// TIA Portal V20 program export: 0 tag tables, 2 data types, 3 data blocks, 7 code blocks (in call order from the OBs), 3 instance data blocks

TYPE "UDT_PusherIO"
// stored: IsFailsafeCompliant false
   STRUCT
      "Step" : Int;
      Fitted : Bool;
      Enable : Bool;
      Mode : Int;
      HopperHighLevel : Bool;
      ManualCycleCmd : Bool;
      JogExtendCmd : Bool;
      JogRetractCmd : Bool;
      HomeLimit : Bool;
      FullTravelLimit : Bool;
      HighPressure : Bool;
      PowerPackRunningFB : Bool;
      FaultReset : Bool;
      EndTravelTimeout : Real;
      ParkedTimeout : Real;
      EndTravelHoldTime : Real;
      PumpRunOnTime : Real;
      JogWarningTime : Real;
      PressureTripConfirmTime : Real;
      PressureClearResumeDelay : Real;
      PressureTripCountThreshold : Int;
      Cycling : Bool;
      Blocked : Bool;
      EndTravelTimeoutFault : Bool;
      ParkedTimeoutFault : Bool;
      BothSwitchesFault : Bool;
      RunPowerPack : Bool;
      Extend : Bool;
      Retract : Bool;
      JogPreStartSounder : Bool;
   END_STRUCT;
END_TYPE

TYPE "UDT_ShredderSequencerIO"
// stored: IsFailsafeCompliant false
   STRUCT
      CycleStart : Bool;
      CycleStop : Bool;
      DownstreamRunning : Bool;
      DischargeConvRunning : Bool;
      HopperLevelHigh : Bool;
      ShredderRunFwdFB : Bool;
      ShredderMotorCurrent : Real;
      MotorFaultActive : Bool;
      FaultReset : Bool;
      OperatorPusherMode : Int;
      PusherJogPreStartSounder : Bool;
      "Step" : Int;
      DischargeConveyorTimeoutFault : Bool;
      ShredderBlockedFault : Bool;
      RunDischargeConv : Bool;
      RunInfeedConv : Bool;
      EnableUpstream : Bool;
      PreStartSounder : Bool;
      InCycle : Bool;
      MotorReverseCmd : Bool;
      MotorAutoStartCmd : Bool;
      MotorPreStartDoneCmd : Bool;
      PusherModeCmd : Int;
   END_STRUCT;
END_TYPE

DATA_BLOCK "DB_Alarms"   // DB5
{ S7_Optimized_Access := 'TRUE' }
VERSION : 0.1
// Category alarms packed per Word (C-501). Bits written by FC_AlarmsMain via documented slice-access exception to C-301.
// stored: AutoNumber true, DBAccessibleFromOPCUA true, IsOnlyStoredInLoadMemory false, IsRetainMemResEnabled false, IsWriteProtectedInAS false, MemoryReserve 100
   VAR
      ShredderAlarm0 : Word;
   END_VAR
BEGIN
END_DATA_BLOCK

DATA_BLOCK "DB_Output"   // DB2
{ S7_Optimized_Access := 'TRUE' }
VERSION : 0.1
// stored: AutoNumber true, DBAccessibleFromOPCUA true, IsOnlyStoredInLoadMemory false, IsRetainMemResEnabled false, IsWriteProtectedInAS false, MemoryReserve 100
   VAR
      Test : Array[0..18] of Bool;
      SpareDQ : Array[1..7] of Bool;
      Run_Shredder_Fwd : Bool;
      Run_Shredder_Rev : Bool;
      Run_PowerPack : Bool;
      Run_Infeed_Conv : Bool;
      Run_Discharge_Conv : Bool;
      Pusher_Extend : Bool;
      Pusher_Retract : Bool;
      In_Cycle : Bool;
      Enable_Upstream : Bool;
      PreStart_Sounder : Bool;
      Motor_Fault_Reset : Bool;
   END_VAR
BEGIN
END_DATA_BLOCK

DATA_BLOCK "DB_Settings"   // DB3
{ S7_Optimized_Access := 'TRUE' }
VERSION : 0.1
// Plant/system-level tunables (C-307) - HMI/operator writes, PLC read-only (C-308). Start values are commissioning defaults (C-309). Members with no start value shown are genuinely unconfigured pending real numbers from the project owner - see the presented build notes, not a guess.
// stored: AutoNumber true, DBAccessibleFromOPCUA true, IsOnlyStoredInLoadMemory false, IsRetainMemResEnabled false, IsWriteProtectedInAS false, MemoryReserve 100
   VAR RETAIN
      PreStartSounderTime : Real := 10.0;
      ShredderReverseRunTime : Real := 6.0;
      InfeedRestartDelay : Real := 5.0;
      InfeedToUpstreamEnableDelay : Real := 3.0;
      OvercurrentSetpointMedium : Real;
      OvercurrentSetpointHigh : Real;
      OvercurrentMediumDelay : Real;
      OvercurrentHighDelay : Real;
      OvercurrentSpinUpAllowance : Real := 3.0;
      ReversalRetryPauseTime : Real := 4.0;
      ReversalWindowTime : Real := 180.0;
      ReversalCountThreshold : Int := 5;
      PressureTripConfirmTime : Real := 0.5;
      PressureClearResumeDelay : Real;
      PressureTripCountThreshold : Int := 5;
      PusherEndTravelTimeout : Real;
      PusherParkedTimeout : Real;
      PusherEndTravelHoldTime : Real := 2.0;
      PusherPumpRunOnTime : Real;
      PusherJogWarningTime : Real := 1.0;
      PusherFitted : Bool := TRUE;
      DischargeConveyorTimeout : Real;
   END_VAR
BEGIN
END_DATA_BLOCK

ORGANIZATION_BLOCK "Main"   // OB1, LAD, ProgramCycle
TITLE = "Main Program Sweep (Cycle)"
{ S7_Optimized_Access := 'TRUE' }
VERSION : 0.1
// stored: AutoNumber true, IsIECCheckEnabled false, SetENOAutomatically false
   VAR_INPUT
      Initial_Call : Bool;   // Initial call of this OB
      Remanence : Bool;   // =True, if remanent data are available
   END_VAR
BEGIN

REGION Network 1: Input Mapping
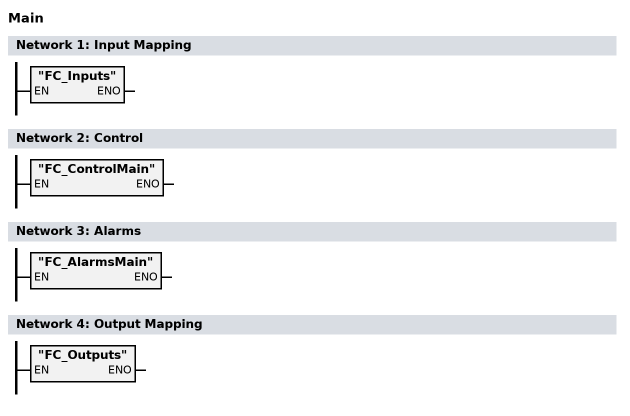
   RUNG wire#powerrail
      "FC_Inputs"()
   END_RUNG
   // the same network as SCL:
   "FC_Inputs"();
END_REGION

REGION Network 2: Control
   RUNG wire#powerrail
      "FC_ControlMain"()
   END_RUNG
   // the same network as SCL:
   "FC_ControlMain"();
END_REGION

REGION Network 3: Alarms
   RUNG wire#powerrail
      "FC_AlarmsMain"()
   END_RUNG
   // the same network as SCL:
   "FC_AlarmsMain"();
END_REGION

REGION Network 4: Output Mapping
   RUNG wire#powerrail
      "FC_Outputs"()
   END_RUNG
   // the same network as SCL:
   "FC_Outputs"();
END_REGION
END_ORGANIZATION_BLOCK

FUNCTION "FC_Inputs" : Void   // FC1, LAD
TITLE = Input Map
{ S7_Optimized_Access := 'TRUE' }
VERSION : 0.1
// stored: AutoNumber true, IsIECCheckEnabled false, SetENOAutomatically false, UDAEnableTagReadback false
BEGIN

REGION Network 1: PLC1 Built-in DI (CPU 1214C)
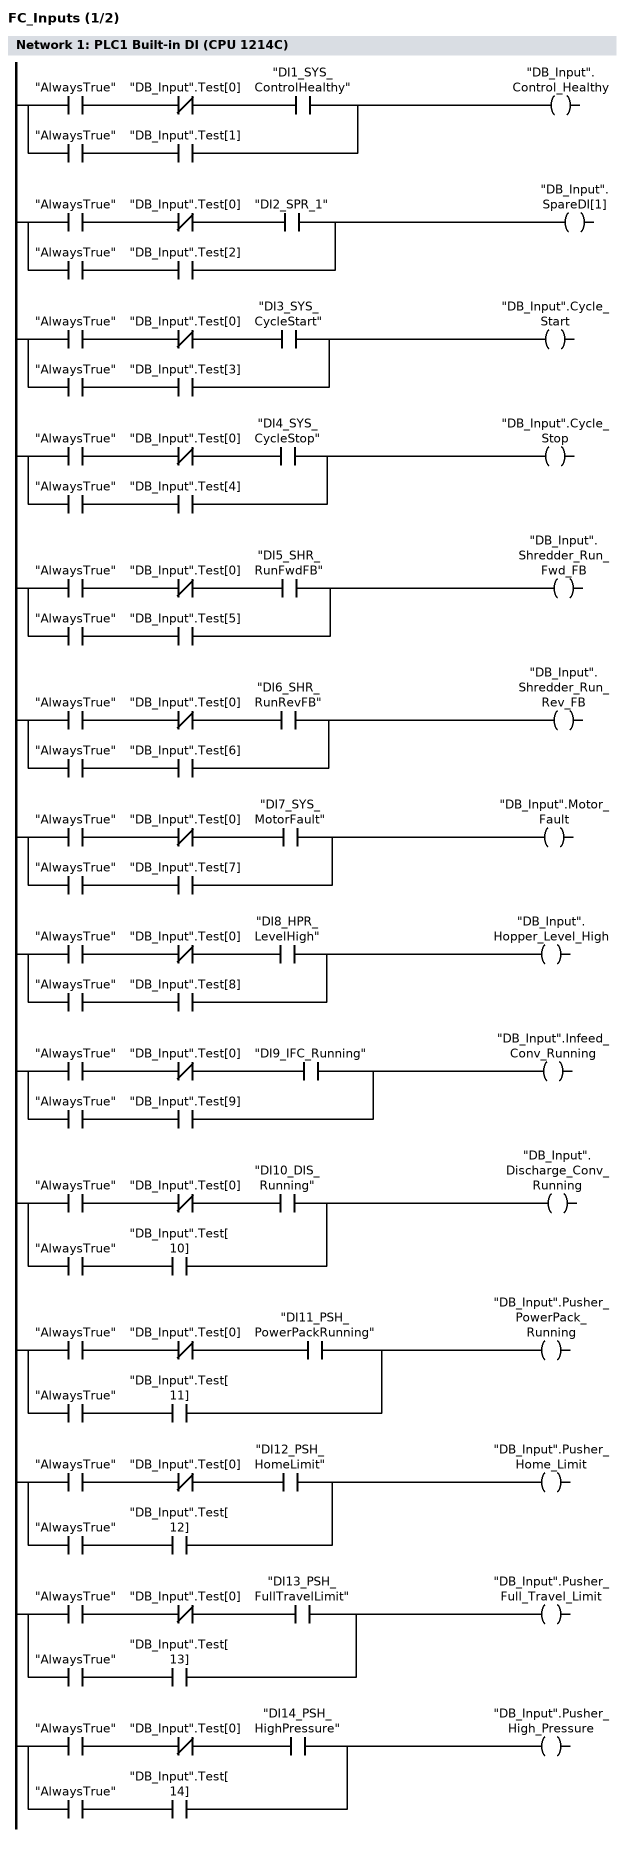
   RUNG wire#powerrail
      Contact( "AlwaysTrue" )
      I_Contact( "DB_Input".Test[0] )
      Contact( "DI1_SYS_ControlHealthy" )
      wire#w1
      Coil( "DB_Input".Control_Healthy )
   END_RUNG
   RUNG wire#powerrail
      Contact( "AlwaysTrue" )
      Contact( "DB_Input".Test[1] )
   END_RUNG wire#w1
   RUNG wire#powerrail
      Contact( "AlwaysTrue" )
      I_Contact( "DB_Input".Test[0] )
      Contact( "DI2_SPR_1" )
      wire#w2
      Coil( "DB_Input".SpareDI[1] )
   END_RUNG
   RUNG wire#powerrail
      Contact( "AlwaysTrue" )
      Contact( "DB_Input".Test[2] )
   END_RUNG wire#w2
   RUNG wire#powerrail
      Contact( "AlwaysTrue" )
      I_Contact( "DB_Input".Test[0] )
      Contact( "DI3_SYS_CycleStart" )
      wire#w3
      Coil( "DB_Input".Cycle_Start )
   END_RUNG
   RUNG wire#powerrail
      Contact( "AlwaysTrue" )
      Contact( "DB_Input".Test[3] )
   END_RUNG wire#w3
   RUNG wire#powerrail
      Contact( "AlwaysTrue" )
      I_Contact( "DB_Input".Test[0] )
      Contact( "DI4_SYS_CycleStop" )
      wire#w4
      Coil( "DB_Input".Cycle_Stop )
   END_RUNG
   RUNG wire#powerrail
      Contact( "AlwaysTrue" )
      Contact( "DB_Input".Test[4] )
   END_RUNG wire#w4
   RUNG wire#powerrail
      Contact( "AlwaysTrue" )
      I_Contact( "DB_Input".Test[0] )
      Contact( "DI5_SHR_RunFwdFB" )
      wire#w5
      Coil( "DB_Input".Shredder_Run_Fwd_FB )
   END_RUNG
   RUNG wire#powerrail
      Contact( "AlwaysTrue" )
      Contact( "DB_Input".Test[5] )
   END_RUNG wire#w5
   RUNG wire#powerrail
      Contact( "AlwaysTrue" )
      I_Contact( "DB_Input".Test[0] )
      Contact( "DI6_SHR_RunRevFB" )
      wire#w6
      Coil( "DB_Input".Shredder_Run_Rev_FB )
   END_RUNG
   RUNG wire#powerrail
      Contact( "AlwaysTrue" )
      Contact( "DB_Input".Test[6] )
   END_RUNG wire#w6
   RUNG wire#powerrail
      Contact( "AlwaysTrue" )
      I_Contact( "DB_Input".Test[0] )
      Contact( "DI7_SYS_MotorFault" )
      wire#w7
      Coil( "DB_Input".Motor_Fault )
   END_RUNG
   RUNG wire#powerrail
      Contact( "AlwaysTrue" )
      Contact( "DB_Input".Test[7] )
   END_RUNG wire#w7
   RUNG wire#powerrail
      Contact( "AlwaysTrue" )
      I_Contact( "DB_Input".Test[0] )
      Contact( "DI8_HPR_LevelHigh" )
      wire#w8
      Coil( "DB_Input".Hopper_Level_High )
   END_RUNG
   RUNG wire#powerrail
      Contact( "AlwaysTrue" )
      Contact( "DB_Input".Test[8] )
   END_RUNG wire#w8
   RUNG wire#powerrail
      Contact( "AlwaysTrue" )
      I_Contact( "DB_Input".Test[0] )
      Contact( "DI9_IFC_Running" )
      wire#w9
      Coil( "DB_Input".Infeed_Conv_Running )
   END_RUNG
   RUNG wire#powerrail
      Contact( "AlwaysTrue" )
      Contact( "DB_Input".Test[9] )
   END_RUNG wire#w9
   RUNG wire#powerrail
      Contact( "AlwaysTrue" )
      I_Contact( "DB_Input".Test[0] )
      Contact( "DI10_DIS_Running" )
      wire#w10
      Coil( "DB_Input".Discharge_Conv_Running )
   END_RUNG
   RUNG wire#powerrail
      Contact( "AlwaysTrue" )
      Contact( "DB_Input".Test[10] )
   END_RUNG wire#w10
   RUNG wire#powerrail
      Contact( "AlwaysTrue" )
      I_Contact( "DB_Input".Test[0] )
      Contact( "DI11_PSH_PowerPackRunning" )
      wire#w11
      Coil( "DB_Input".Pusher_PowerPack_Running )
   END_RUNG
   RUNG wire#powerrail
      Contact( "AlwaysTrue" )
      Contact( "DB_Input".Test[11] )
   END_RUNG wire#w11
   RUNG wire#powerrail
      Contact( "AlwaysTrue" )
      I_Contact( "DB_Input".Test[0] )
      Contact( "DI12_PSH_HomeLimit" )
      wire#w12
      Coil( "DB_Input".Pusher_Home_Limit )
   END_RUNG
   RUNG wire#powerrail
      Contact( "AlwaysTrue" )
      Contact( "DB_Input".Test[12] )
   END_RUNG wire#w12
   RUNG wire#powerrail
      Contact( "AlwaysTrue" )
      I_Contact( "DB_Input".Test[0] )
      Contact( "DI13_PSH_FullTravelLimit" )
      wire#w13
      Coil( "DB_Input".Pusher_Full_Travel_Limit )
   END_RUNG
   RUNG wire#powerrail
      Contact( "AlwaysTrue" )
      Contact( "DB_Input".Test[13] )
   END_RUNG wire#w13
   RUNG wire#powerrail
      Contact( "AlwaysTrue" )
      I_Contact( "DB_Input".Test[0] )
      Contact( "DI14_PSH_HighPressure" )
      wire#w14
      Coil( "DB_Input".Pusher_High_Pressure )
   END_RUNG
   RUNG wire#powerrail
      Contact( "AlwaysTrue" )
      Contact( "DB_Input".Test[14] )
   END_RUNG wire#w14
   // the same network as SCL:
   "DB_Input".Control_Healthy := ("AlwaysTrue" AND NOT "DB_Input".Test[0] AND "DI1_SYS_ControlHealthy") OR ("AlwaysTrue" AND "DB_Input".Test[1]);
   "DB_Input".SpareDI[1] := ("AlwaysTrue" AND NOT "DB_Input".Test[0] AND "DI2_SPR_1") OR ("AlwaysTrue" AND "DB_Input".Test[2]);
   "DB_Input".Cycle_Start := ("AlwaysTrue" AND NOT "DB_Input".Test[0] AND "DI3_SYS_CycleStart") OR ("AlwaysTrue" AND "DB_Input".Test[3]);
   "DB_Input".Cycle_Stop := ("AlwaysTrue" AND NOT "DB_Input".Test[0] AND "DI4_SYS_CycleStop") OR ("AlwaysTrue" AND "DB_Input".Test[4]);
   "DB_Input".Shredder_Run_Fwd_FB := ("AlwaysTrue" AND NOT "DB_Input".Test[0] AND "DI5_SHR_RunFwdFB") OR ("AlwaysTrue" AND "DB_Input".Test[5]);
   "DB_Input".Shredder_Run_Rev_FB := ("AlwaysTrue" AND NOT "DB_Input".Test[0] AND "DI6_SHR_RunRevFB") OR ("AlwaysTrue" AND "DB_Input".Test[6]);
   "DB_Input".Motor_Fault := ("AlwaysTrue" AND NOT "DB_Input".Test[0] AND "DI7_SYS_MotorFault") OR ("AlwaysTrue" AND "DB_Input".Test[7]);
   "DB_Input".Hopper_Level_High := ("AlwaysTrue" AND NOT "DB_Input".Test[0] AND "DI8_HPR_LevelHigh") OR ("AlwaysTrue" AND "DB_Input".Test[8]);
   "DB_Input".Infeed_Conv_Running := ("AlwaysTrue" AND NOT "DB_Input".Test[0] AND "DI9_IFC_Running") OR ("AlwaysTrue" AND "DB_Input".Test[9]);
   "DB_Input".Discharge_Conv_Running := ("AlwaysTrue" AND NOT "DB_Input".Test[0] AND "DI10_DIS_Running") OR ("AlwaysTrue" AND "DB_Input".Test[10]);
   "DB_Input".Pusher_PowerPack_Running := ("AlwaysTrue" AND NOT "DB_Input".Test[0] AND "DI11_PSH_PowerPackRunning") OR ("AlwaysTrue" AND "DB_Input".Test[11]);
   "DB_Input".Pusher_Home_Limit := ("AlwaysTrue" AND NOT "DB_Input".Test[0] AND "DI12_PSH_HomeLimit") OR ("AlwaysTrue" AND "DB_Input".Test[12]);
   "DB_Input".Pusher_Full_Travel_Limit := ("AlwaysTrue" AND NOT "DB_Input".Test[0] AND "DI13_PSH_FullTravelLimit") OR ("AlwaysTrue" AND "DB_Input".Test[13]);
   "DB_Input".Pusher_High_Pressure := ("AlwaysTrue" AND NOT "DB_Input".Test[0] AND "DI14_PSH_HighPressure") OR ("AlwaysTrue" AND "DB_Input".Test[14]);
END_REGION

REGION Network 2: PLC1.1 SM1223 DI
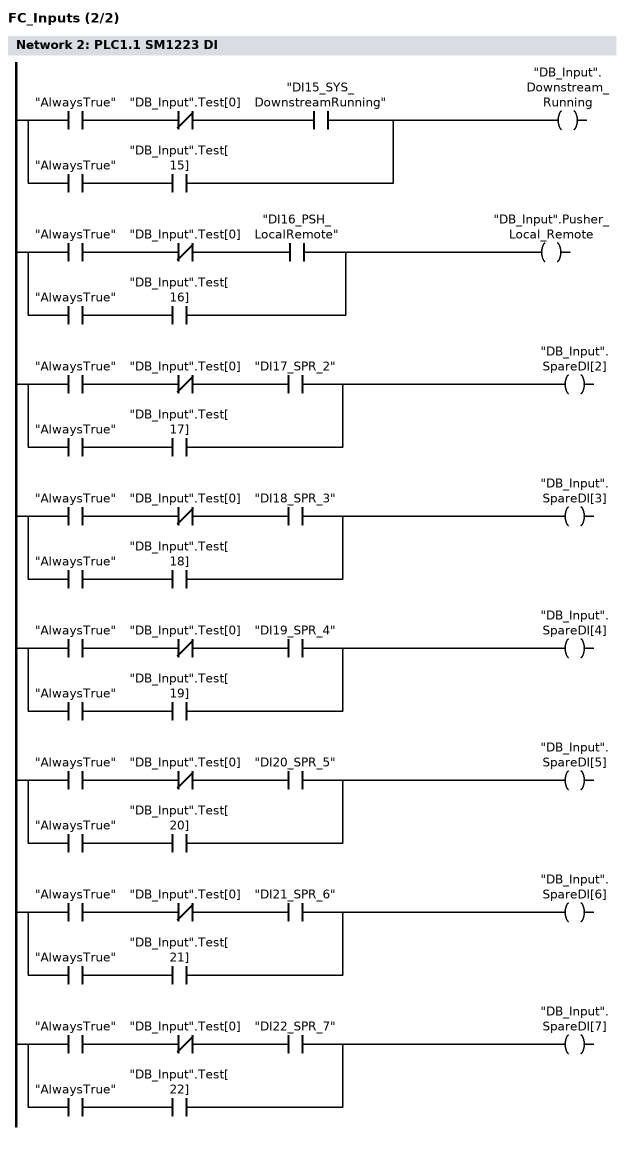
   RUNG wire#powerrail
      Contact( "AlwaysTrue" )
      I_Contact( "DB_Input".Test[0] )
      Contact( "DI15_SYS_DownstreamRunning" )
      wire#w1
      Coil( "DB_Input".Downstream_Running )
   END_RUNG
   RUNG wire#powerrail
      Contact( "AlwaysTrue" )
      Contact( "DB_Input".Test[15] )
   END_RUNG wire#w1
   RUNG wire#powerrail
      Contact( "AlwaysTrue" )
      I_Contact( "DB_Input".Test[0] )
      Contact( "DI16_PSH_LocalRemote" )
      wire#w2
      Coil( "DB_Input".Pusher_Local_Remote )
   END_RUNG
   RUNG wire#powerrail
      Contact( "AlwaysTrue" )
      Contact( "DB_Input".Test[16] )
   END_RUNG wire#w2
   RUNG wire#powerrail
      Contact( "AlwaysTrue" )
      I_Contact( "DB_Input".Test[0] )
      Contact( "DI17_SPR_2" )
      wire#w3
      Coil( "DB_Input".SpareDI[2] )
   END_RUNG
   RUNG wire#powerrail
      Contact( "AlwaysTrue" )
      Contact( "DB_Input".Test[17] )
   END_RUNG wire#w3
   RUNG wire#powerrail
      Contact( "AlwaysTrue" )
      I_Contact( "DB_Input".Test[0] )
      Contact( "DI18_SPR_3" )
      wire#w4
      Coil( "DB_Input".SpareDI[3] )
   END_RUNG
   RUNG wire#powerrail
      Contact( "AlwaysTrue" )
      Contact( "DB_Input".Test[18] )
   END_RUNG wire#w4
   RUNG wire#powerrail
      Contact( "AlwaysTrue" )
      I_Contact( "DB_Input".Test[0] )
      Contact( "DI19_SPR_4" )
      wire#w5
      Coil( "DB_Input".SpareDI[4] )
   END_RUNG
   RUNG wire#powerrail
      Contact( "AlwaysTrue" )
      Contact( "DB_Input".Test[19] )
   END_RUNG wire#w5
   RUNG wire#powerrail
      Contact( "AlwaysTrue" )
      I_Contact( "DB_Input".Test[0] )
      Contact( "DI20_SPR_5" )
      wire#w6
      Coil( "DB_Input".SpareDI[5] )
   END_RUNG
   RUNG wire#powerrail
      Contact( "AlwaysTrue" )
      Contact( "DB_Input".Test[20] )
   END_RUNG wire#w6
   RUNG wire#powerrail
      Contact( "AlwaysTrue" )
      I_Contact( "DB_Input".Test[0] )
      Contact( "DI21_SPR_6" )
      wire#w7
      Coil( "DB_Input".SpareDI[6] )
   END_RUNG
   RUNG wire#powerrail
      Contact( "AlwaysTrue" )
      Contact( "DB_Input".Test[21] )
   END_RUNG wire#w7
   RUNG wire#powerrail
      Contact( "AlwaysTrue" )
      I_Contact( "DB_Input".Test[0] )
      Contact( "DI22_SPR_7" )
      wire#w8
      Coil( "DB_Input".SpareDI[7] )
   END_RUNG
   RUNG wire#powerrail
      Contact( "AlwaysTrue" )
      Contact( "DB_Input".Test[22] )
   END_RUNG wire#w8
   // the same network as SCL:
   "DB_Input".Downstream_Running := ("AlwaysTrue" AND NOT "DB_Input".Test[0] AND "DI15_SYS_DownstreamRunning") OR ("AlwaysTrue" AND "DB_Input".Test[15]);
   "DB_Input".Pusher_Local_Remote := ("AlwaysTrue" AND NOT "DB_Input".Test[0] AND "DI16_PSH_LocalRemote") OR ("AlwaysTrue" AND "DB_Input".Test[16]);
   "DB_Input".SpareDI[2] := ("AlwaysTrue" AND NOT "DB_Input".Test[0] AND "DI17_SPR_2") OR ("AlwaysTrue" AND "DB_Input".Test[17]);
   "DB_Input".SpareDI[3] := ("AlwaysTrue" AND NOT "DB_Input".Test[0] AND "DI18_SPR_3") OR ("AlwaysTrue" AND "DB_Input".Test[18]);
   "DB_Input".SpareDI[4] := ("AlwaysTrue" AND NOT "DB_Input".Test[0] AND "DI19_SPR_4") OR ("AlwaysTrue" AND "DB_Input".Test[19]);
   "DB_Input".SpareDI[5] := ("AlwaysTrue" AND NOT "DB_Input".Test[0] AND "DI20_SPR_5") OR ("AlwaysTrue" AND "DB_Input".Test[20]);
   "DB_Input".SpareDI[6] := ("AlwaysTrue" AND NOT "DB_Input".Test[0] AND "DI21_SPR_6") OR ("AlwaysTrue" AND "DB_Input".Test[21]);
   "DB_Input".SpareDI[7] := ("AlwaysTrue" AND NOT "DB_Input".Test[0] AND "DI22_SPR_7") OR ("AlwaysTrue" AND "DB_Input".Test[22]);
END_REGION
END_FUNCTION

FUNCTION "FC_ControlMain" : Void   // FC3, LAD
TITLE = Control Main
{ S7_Optimized_Access := 'TRUE' }
VERSION : 0.1
// stored: AutoNumber true, IsIECCheckEnabled false, SetENOAutomatically false, UDAEnableTagReadback false
BEGIN

REGION Network 1: Sequencer Input Wiring
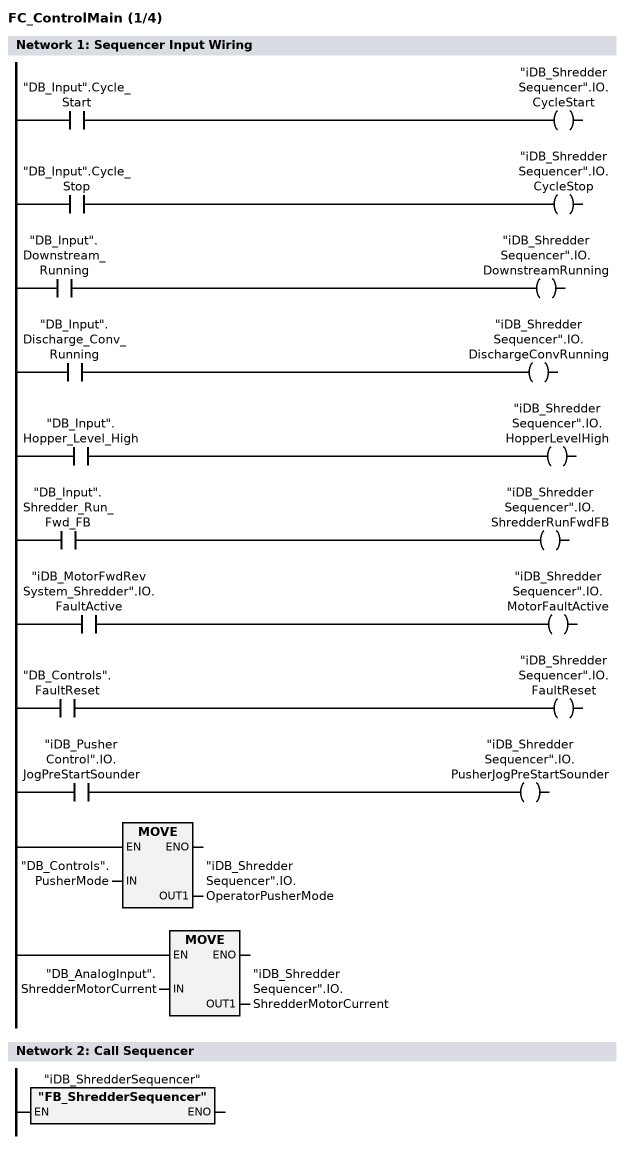
   RUNG wire#powerrail
      Contact( "DB_Input".Cycle_Start )
      Coil( "iDB_ShredderSequencer".IO.CycleStart )
   END_RUNG
   RUNG wire#powerrail
      Contact( "DB_Input".Cycle_Stop )
      Coil( "iDB_ShredderSequencer".IO.CycleStop )
   END_RUNG
   RUNG wire#powerrail
      Contact( "DB_Input".Downstream_Running )
      Coil( "iDB_ShredderSequencer".IO.DownstreamRunning )
   END_RUNG
   RUNG wire#powerrail
      Contact( "DB_Input".Discharge_Conv_Running )
      Coil( "iDB_ShredderSequencer".IO.DischargeConvRunning )
   END_RUNG
   RUNG wire#powerrail
      Contact( "DB_Input".Hopper_Level_High )
      Coil( "iDB_ShredderSequencer".IO.HopperLevelHigh )
   END_RUNG
   RUNG wire#powerrail
      Contact( "DB_Input".Shredder_Run_Fwd_FB )
      Coil( "iDB_ShredderSequencer".IO.ShredderRunFwdFB )
   END_RUNG
   RUNG wire#powerrail
      Contact( "iDB_MotorFwdRevSystem_Shredder".IO.FaultActive )
      Coil( "iDB_ShredderSequencer".IO.MotorFaultActive )
   END_RUNG
   RUNG wire#powerrail
      Contact( "DB_Controls".FaultReset )
      Coil( "iDB_ShredderSequencer".IO.FaultReset )
   END_RUNG
   RUNG wire#powerrail
      Contact( "iDB_PusherControl".IO.JogPreStartSounder )
      Coil( "iDB_ShredderSequencer".IO.PusherJogPreStartSounder )
   END_RUNG
   RUNG wire#powerrail
      Move(in := "DB_Controls".PusherMode, out1 => "iDB_ShredderSequencer".IO.OperatorPusherMode)
   END_RUNG
   RUNG wire#powerrail
      Move(in := "DB_AnalogInput".ShredderMotorCurrent, out1 => "iDB_ShredderSequencer".IO.ShredderMotorCurrent)
   END_RUNG
   // the same network as SCL:
   "iDB_ShredderSequencer".IO.CycleStart := "DB_Input".Cycle_Start;
   "iDB_ShredderSequencer".IO.CycleStop := "DB_Input".Cycle_Stop;
   "iDB_ShredderSequencer".IO.DownstreamRunning := "DB_Input".Downstream_Running;
   "iDB_ShredderSequencer".IO.DischargeConvRunning := "DB_Input".Discharge_Conv_Running;
   "iDB_ShredderSequencer".IO.HopperLevelHigh := "DB_Input".Hopper_Level_High;
   "iDB_ShredderSequencer".IO.ShredderRunFwdFB := "DB_Input".Shredder_Run_Fwd_FB;
   "iDB_ShredderSequencer".IO.MotorFaultActive := "iDB_MotorFwdRevSystem_Shredder".IO.FaultActive;
   "iDB_ShredderSequencer".IO.FaultReset := "DB_Controls".FaultReset;
   "iDB_ShredderSequencer".IO.PusherJogPreStartSounder := "iDB_PusherControl".IO.JogPreStartSounder;
   "iDB_ShredderSequencer".IO.OperatorPusherMode := "DB_Controls".PusherMode;
   "iDB_ShredderSequencer".IO.ShredderMotorCurrent := "DB_AnalogInput".ShredderMotorCurrent;
END_REGION

REGION Network 2: Call Sequencer
   RUNG wire#powerrail
      "iDB_ShredderSequencer"()
   END_RUNG
   // the same network as SCL:
   "iDB_ShredderSequencer"();   // "FB_ShredderSequencer"
END_REGION

REGION Network 3: MotorFwdRevSystem Wiring
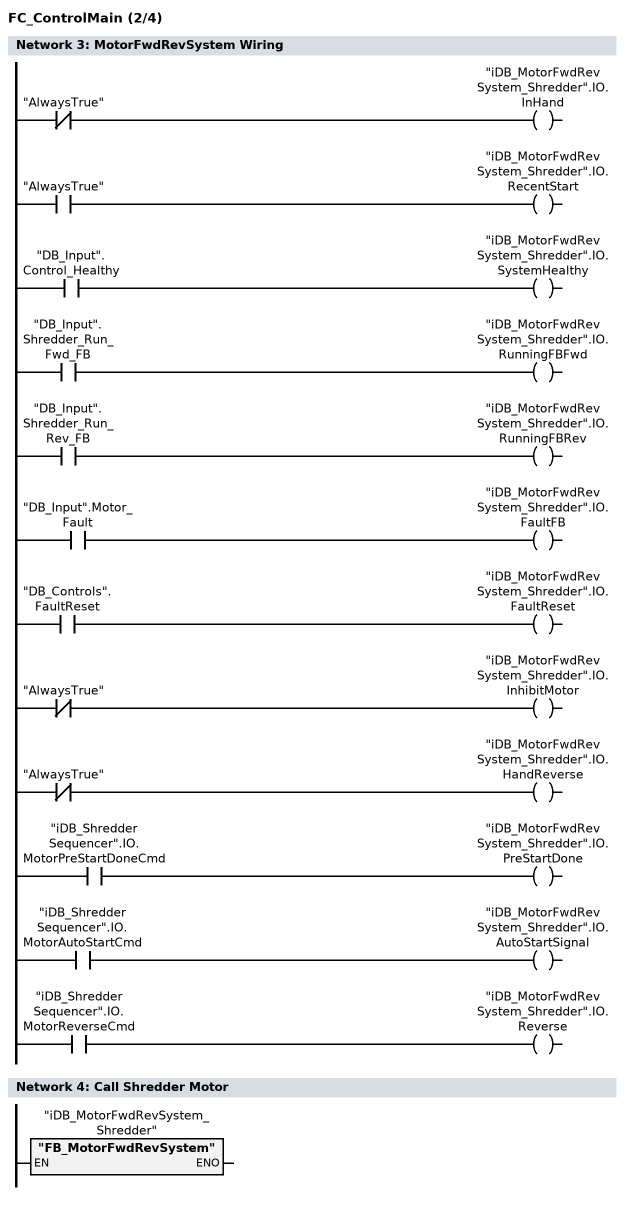
   RUNG wire#powerrail
      I_Contact( "AlwaysTrue" )
      Coil( "iDB_MotorFwdRevSystem_Shredder".IO.InHand )
   END_RUNG
   RUNG wire#powerrail
      Contact( "AlwaysTrue" )
      Coil( "iDB_MotorFwdRevSystem_Shredder".IO.RecentStart )
   END_RUNG
   RUNG wire#powerrail
      Contact( "DB_Input".Control_Healthy )
      Coil( "iDB_MotorFwdRevSystem_Shredder".IO.SystemHealthy )
   END_RUNG
   RUNG wire#powerrail
      Contact( "DB_Input".Shredder_Run_Fwd_FB )
      Coil( "iDB_MotorFwdRevSystem_Shredder".IO.RunningFBFwd )
   END_RUNG
   RUNG wire#powerrail
      Contact( "DB_Input".Shredder_Run_Rev_FB )
      Coil( "iDB_MotorFwdRevSystem_Shredder".IO.RunningFBRev )
   END_RUNG
   RUNG wire#powerrail
      Contact( "DB_Input".Motor_Fault )
      Coil( "iDB_MotorFwdRevSystem_Shredder".IO.FaultFB )
   END_RUNG
   RUNG wire#powerrail
      Contact( "DB_Controls".FaultReset )
      Coil( "iDB_MotorFwdRevSystem_Shredder".IO.FaultReset )
   END_RUNG
   RUNG wire#powerrail
      I_Contact( "AlwaysTrue" )
      Coil( "iDB_MotorFwdRevSystem_Shredder".IO.InhibitMotor )
   END_RUNG
   RUNG wire#powerrail
      I_Contact( "AlwaysTrue" )
      Coil( "iDB_MotorFwdRevSystem_Shredder".IO.HandReverse )
   END_RUNG
   RUNG wire#powerrail
      Contact( "iDB_ShredderSequencer".IO.MotorPreStartDoneCmd )
      Coil( "iDB_MotorFwdRevSystem_Shredder".IO.PreStartDone )
   END_RUNG
   RUNG wire#powerrail
      Contact( "iDB_ShredderSequencer".IO.MotorAutoStartCmd )
      Coil( "iDB_MotorFwdRevSystem_Shredder".IO.AutoStartSignal )
   END_RUNG
   RUNG wire#powerrail
      Contact( "iDB_ShredderSequencer".IO.MotorReverseCmd )
      Coil( "iDB_MotorFwdRevSystem_Shredder".IO.Reverse )
   END_RUNG
   // the same network as SCL:
   "iDB_MotorFwdRevSystem_Shredder".IO.InHand := NOT "AlwaysTrue";
   "iDB_MotorFwdRevSystem_Shredder".IO.RecentStart := "AlwaysTrue";
   "iDB_MotorFwdRevSystem_Shredder".IO.SystemHealthy := "DB_Input".Control_Healthy;
   "iDB_MotorFwdRevSystem_Shredder".IO.RunningFBFwd := "DB_Input".Shredder_Run_Fwd_FB;
   "iDB_MotorFwdRevSystem_Shredder".IO.RunningFBRev := "DB_Input".Shredder_Run_Rev_FB;
   "iDB_MotorFwdRevSystem_Shredder".IO.FaultFB := "DB_Input".Motor_Fault;
   "iDB_MotorFwdRevSystem_Shredder".IO.FaultReset := "DB_Controls".FaultReset;
   "iDB_MotorFwdRevSystem_Shredder".IO.InhibitMotor := NOT "AlwaysTrue";
   "iDB_MotorFwdRevSystem_Shredder".IO.HandReverse := NOT "AlwaysTrue";
   "iDB_MotorFwdRevSystem_Shredder".IO.PreStartDone := "iDB_ShredderSequencer".IO.MotorPreStartDoneCmd;
   "iDB_MotorFwdRevSystem_Shredder".IO.AutoStartSignal := "iDB_ShredderSequencer".IO.MotorAutoStartCmd;
   "iDB_MotorFwdRevSystem_Shredder".IO.Reverse := "iDB_ShredderSequencer".IO.MotorReverseCmd;
END_REGION

REGION Network 4: Call Shredder Motor
   RUNG wire#powerrail
      "iDB_MotorFwdRevSystem_Shredder"()
   END_RUNG
   // the same network as SCL:
   "iDB_MotorFwdRevSystem_Shredder"();   // "FB_MotorFwdRevSystem"
END_REGION

REGION Network 5: PusherControl Wiring
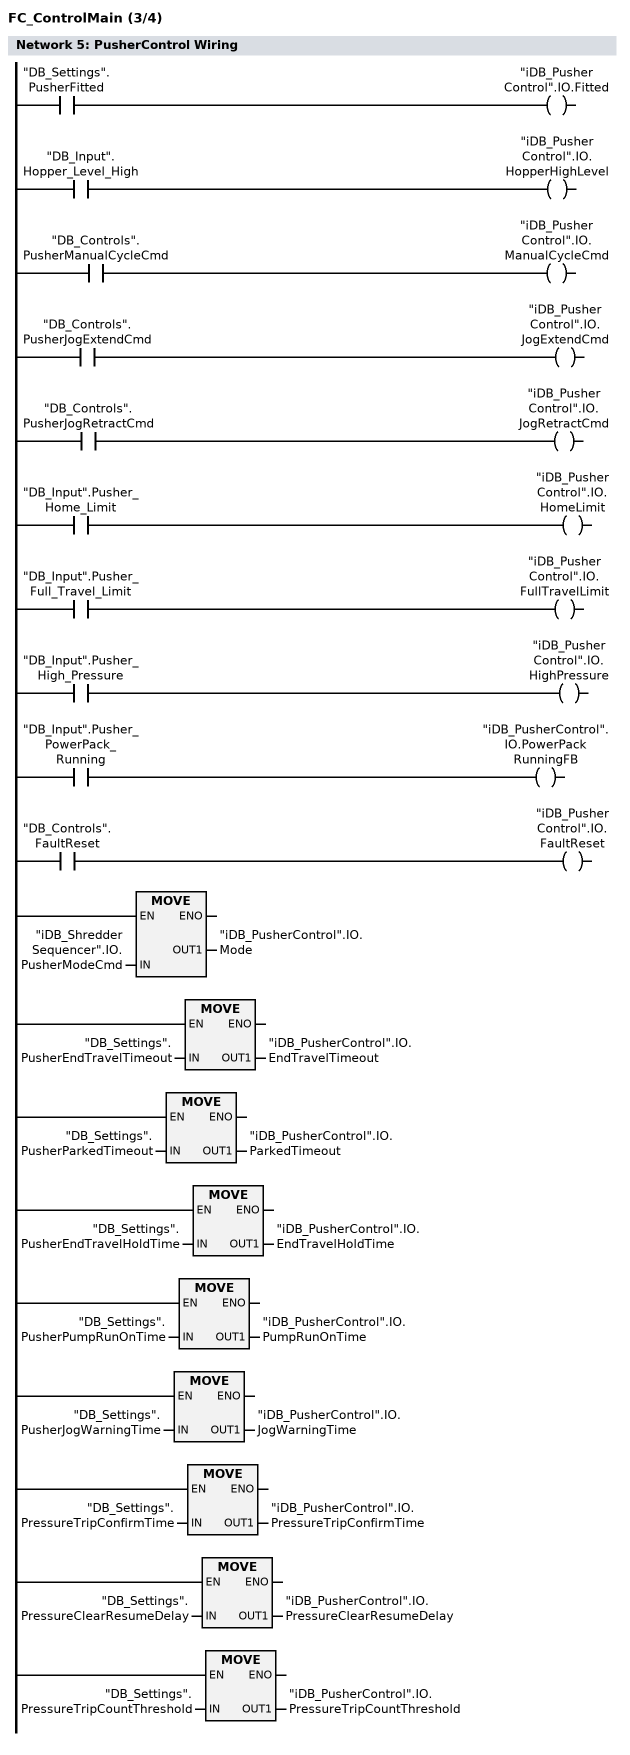
   RUNG wire#powerrail
      Contact( "DB_Settings".PusherFitted )
      Coil( "iDB_PusherControl".IO.Fitted )
   END_RUNG
   RUNG wire#powerrail
      Contact( "DB_Input".Hopper_Level_High )
      Coil( "iDB_PusherControl".IO.HopperHighLevel )
   END_RUNG
   RUNG wire#powerrail
      Contact( "DB_Controls".PusherManualCycleCmd )
      Coil( "iDB_PusherControl".IO.ManualCycleCmd )
   END_RUNG
   RUNG wire#powerrail
      Contact( "DB_Controls".PusherJogExtendCmd )
      Coil( "iDB_PusherControl".IO.JogExtendCmd )
   END_RUNG
   RUNG wire#powerrail
      Contact( "DB_Controls".PusherJogRetractCmd )
      Coil( "iDB_PusherControl".IO.JogRetractCmd )
   END_RUNG
   RUNG wire#powerrail
      Contact( "DB_Input".Pusher_Home_Limit )
      Coil( "iDB_PusherControl".IO.HomeLimit )
   END_RUNG
   RUNG wire#powerrail
      Contact( "DB_Input".Pusher_Full_Travel_Limit )
      Coil( "iDB_PusherControl".IO.FullTravelLimit )
   END_RUNG
   RUNG wire#powerrail
      Contact( "DB_Input".Pusher_High_Pressure )
      Coil( "iDB_PusherControl".IO.HighPressure )
   END_RUNG
   RUNG wire#powerrail
      Contact( "DB_Input".Pusher_PowerPack_Running )
      Coil( "iDB_PusherControl".IO.PowerPackRunningFB )
   END_RUNG
   RUNG wire#powerrail
      Contact( "DB_Controls".FaultReset )
      Coil( "iDB_PusherControl".IO.FaultReset )
   END_RUNG
   RUNG wire#powerrail
      Move(in := "iDB_ShredderSequencer".IO.PusherModeCmd, out1 => "iDB_PusherControl".IO.Mode)
   END_RUNG
   RUNG wire#powerrail
      Move(in := "DB_Settings".PusherEndTravelTimeout, out1 => "iDB_PusherControl".IO.EndTravelTimeout)
   END_RUNG
   RUNG wire#powerrail
      Move(in := "DB_Settings".PusherParkedTimeout, out1 => "iDB_PusherControl".IO.ParkedTimeout)
   END_RUNG
   RUNG wire#powerrail
      Move(in := "DB_Settings".PusherEndTravelHoldTime, out1 => "iDB_PusherControl".IO.EndTravelHoldTime)
   END_RUNG
   RUNG wire#powerrail
      Move(in := "DB_Settings".PusherPumpRunOnTime, out1 => "iDB_PusherControl".IO.PumpRunOnTime)
   END_RUNG
   RUNG wire#powerrail
      Move(in := "DB_Settings".PusherJogWarningTime, out1 => "iDB_PusherControl".IO.JogWarningTime)
   END_RUNG
   RUNG wire#powerrail
      Move(in := "DB_Settings".PressureTripConfirmTime, out1 => "iDB_PusherControl".IO.PressureTripConfirmTime)
   END_RUNG
   RUNG wire#powerrail
      Move(in := "DB_Settings".PressureClearResumeDelay, out1 => "iDB_PusherControl".IO.PressureClearResumeDelay)
   END_RUNG
   RUNG wire#powerrail
      Move(in := "DB_Settings".PressureTripCountThreshold, out1 => "iDB_PusherControl".IO.PressureTripCountThreshold)
   END_RUNG
   // the same network as SCL:
   "iDB_PusherControl".IO.Fitted := "DB_Settings".PusherFitted;
   "iDB_PusherControl".IO.HopperHighLevel := "DB_Input".Hopper_Level_High;
   "iDB_PusherControl".IO.ManualCycleCmd := "DB_Controls".PusherManualCycleCmd;
   "iDB_PusherControl".IO.JogExtendCmd := "DB_Controls".PusherJogExtendCmd;
   "iDB_PusherControl".IO.JogRetractCmd := "DB_Controls".PusherJogRetractCmd;
   "iDB_PusherControl".IO.HomeLimit := "DB_Input".Pusher_Home_Limit;
   "iDB_PusherControl".IO.FullTravelLimit := "DB_Input".Pusher_Full_Travel_Limit;
   "iDB_PusherControl".IO.HighPressure := "DB_Input".Pusher_High_Pressure;
   "iDB_PusherControl".IO.PowerPackRunningFB := "DB_Input".Pusher_PowerPack_Running;
   "iDB_PusherControl".IO.FaultReset := "DB_Controls".FaultReset;
   "iDB_PusherControl".IO.Mode := "iDB_ShredderSequencer".IO.PusherModeCmd;
   "iDB_PusherControl".IO.EndTravelTimeout := "DB_Settings".PusherEndTravelTimeout;
   "iDB_PusherControl".IO.ParkedTimeout := "DB_Settings".PusherParkedTimeout;
   "iDB_PusherControl".IO.EndTravelHoldTime := "DB_Settings".PusherEndTravelHoldTime;
   "iDB_PusherControl".IO.PumpRunOnTime := "DB_Settings".PusherPumpRunOnTime;
   "iDB_PusherControl".IO.JogWarningTime := "DB_Settings".PusherJogWarningTime;
   "iDB_PusherControl".IO.PressureTripConfirmTime := "DB_Settings".PressureTripConfirmTime;
   "iDB_PusherControl".IO.PressureClearResumeDelay := "DB_Settings".PressureClearResumeDelay;
   "iDB_PusherControl".IO.PressureTripCountThreshold := "DB_Settings".PressureTripCountThreshold;
END_REGION

REGION Network 6: Call Pusher
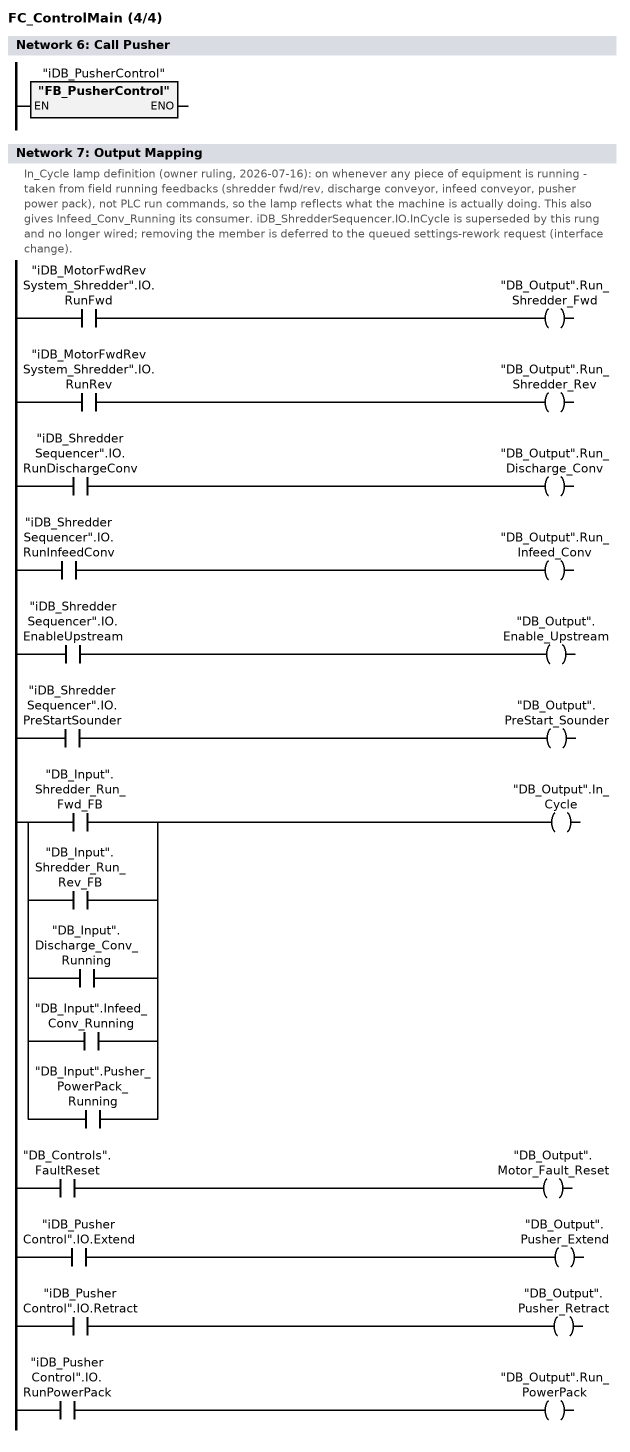
   RUNG wire#powerrail
      "iDB_PusherControl"()
   END_RUNG
   // the same network as SCL:
   "iDB_PusherControl"();   // "FB_PusherControl"
END_REGION

REGION Network 7: Output Mapping
   // In_Cycle lamp definition (owner ruling, 2026-07-16): on whenever any piece of equipment is running - taken from field running feedbacks (shredder fwd/rev, discharge conveyor, infeed conveyor, pusher power pack), not PLC run commands, so the lamp reflects what the machine is actually doing. This also gives Infeed_Conv_Running its consumer. iDB_ShredderSequencer.IO.InCycle is superseded by this rung and no longer wired; removing the member is deferred to the queued settings-rework request (interface change).
   RUNG wire#powerrail
      Contact( "iDB_MotorFwdRevSystem_Shredder".IO.RunFwd )
      Coil( "DB_Output".Run_Shredder_Fwd )
   END_RUNG
   RUNG wire#powerrail
      Contact( "iDB_MotorFwdRevSystem_Shredder".IO.RunRev )
      Coil( "DB_Output".Run_Shredder_Rev )
   END_RUNG
   RUNG wire#powerrail
      Contact( "iDB_ShredderSequencer".IO.RunDischargeConv )
      Coil( "DB_Output".Run_Discharge_Conv )
   END_RUNG
   RUNG wire#powerrail
      Contact( "iDB_ShredderSequencer".IO.RunInfeedConv )
      Coil( "DB_Output".Run_Infeed_Conv )
   END_RUNG
   RUNG wire#powerrail
      Contact( "iDB_ShredderSequencer".IO.EnableUpstream )
      Coil( "DB_Output".Enable_Upstream )
   END_RUNG
   RUNG wire#powerrail
      Contact( "iDB_ShredderSequencer".IO.PreStartSounder )
      Coil( "DB_Output".PreStart_Sounder )
   END_RUNG
   RUNG wire#powerrail
      Contact( "DB_Input".Shredder_Run_Fwd_FB )
      wire#w1
      Coil( "DB_Output".In_Cycle )
   END_RUNG
   RUNG wire#powerrail
      Contact( "DB_Input".Shredder_Run_Rev_FB )
   END_RUNG wire#w1
   RUNG wire#powerrail
      Contact( "DB_Input".Discharge_Conv_Running )
   END_RUNG wire#w1
   RUNG wire#powerrail
      Contact( "DB_Input".Infeed_Conv_Running )
   END_RUNG wire#w1
   RUNG wire#powerrail
      Contact( "DB_Input".Pusher_PowerPack_Running )
   END_RUNG wire#w1
   RUNG wire#powerrail
      Contact( "DB_Controls".FaultReset )
      Coil( "DB_Output".Motor_Fault_Reset )
   END_RUNG
   RUNG wire#powerrail
      Contact( "iDB_PusherControl".IO.Extend )
      Coil( "DB_Output".Pusher_Extend )
   END_RUNG
   RUNG wire#powerrail
      Contact( "iDB_PusherControl".IO.Retract )
      Coil( "DB_Output".Pusher_Retract )
   END_RUNG
   RUNG wire#powerrail
      Contact( "iDB_PusherControl".IO.RunPowerPack )
      Coil( "DB_Output".Run_PowerPack )
   END_RUNG
   // the same network as SCL:
   "DB_Output".Run_Shredder_Fwd := "iDB_MotorFwdRevSystem_Shredder".IO.RunFwd;
   "DB_Output".Run_Shredder_Rev := "iDB_MotorFwdRevSystem_Shredder".IO.RunRev;
   "DB_Output".Run_Discharge_Conv := "iDB_ShredderSequencer".IO.RunDischargeConv;
   "DB_Output".Run_Infeed_Conv := "iDB_ShredderSequencer".IO.RunInfeedConv;
   "DB_Output".Enable_Upstream := "iDB_ShredderSequencer".IO.EnableUpstream;
   "DB_Output".PreStart_Sounder := "iDB_ShredderSequencer".IO.PreStartSounder;
   "DB_Output".In_Cycle := "DB_Input".Shredder_Run_Fwd_FB OR "DB_Input".Shredder_Run_Rev_FB OR "DB_Input".Discharge_Conv_Running OR "DB_Input".Infeed_Conv_Running OR "DB_Input".Pusher_PowerPack_Running;
   "DB_Output".Motor_Fault_Reset := "DB_Controls".FaultReset;
   "DB_Output".Pusher_Extend := "iDB_PusherControl".IO.Extend;
   "DB_Output".Pusher_Retract := "iDB_PusherControl".IO.Retract;
   "DB_Output".Run_PowerPack := "iDB_PusherControl".IO.RunPowerPack;
END_REGION
END_FUNCTION

FUNCTION_BLOCK "FB_ShredderSequencer"   // FB8, LAD
TITLE = Shredder Plant Sequencer
{ S7_Optimized_Access := 'TRUE' }
VERSION : 0.1
// Shredder plant sequencer (C-118-C-125): commands the shredder motor (via FB_MotorFwdRevSystem, wired at FC_ControlMain) and gates infeed/discharge conveyors and upstream enable, through a stepped cycle. Step legend (C-120): 0=Idle (stopped, waiting for a start condition) - 10=PreStart (siren warning before motion) - 20=DischargeStart (discharge conveyor starting, timed) - 30=ReverseRun (shredder commanded reverse - see FB_MotorFwdRevSystem's own pause/reversal handling) - 40=WaitForwardRun (waiting for forward-run feedback) - 50=Running (normal production; infeed/upstream-enable timers and overcurrent detection are live) - 60=OvercurrentAbort (tripped - pause, then retry into ReverseRun, or stay out if too many reversals).
// stored: AutoNumber true, IsIECCheckEnabled false, IsRetainMemResEnabled false, MemoryReserve 100, SetENOAutomatically false, UDAEnableTagReadback false
   VAR RETAIN
      IO { S7_SetPoint := 'True'} : "UDT_ShredderSequencerIO";   // Caller-visible interface (C-115) - FC_ControlMain writes CycleStart/CycleStop/feedback/tunables in, reads Run*/EnableUpstream/PreStartSounder/motor-command bits out. See the block header for the Step value legend.
   END_VAR
   VAR
      StopCmd : Bool;   // Loss of DownstreamRunning stops the shredder too, not just an operator CycleStop - nowhere for shredded material to go otherwise. Read by every step's own stop transition below.
      ReversalWindowTimeMS : DInt;
      PreStartSounderTimeMS : DInt;
      DischargeConveyorTimeoutMS : DInt;
      ShredderReverseRunTimeMS : DInt;
      InfeedRestartDelayMS : DInt;
      InfeedToUpstreamEnableDelayMS : DInt;
      OvercurrentSpinUpAllowanceMS : DInt;
      OvercurrentMediumDelayMS : DInt;
      OvercurrentHighDelayMS : DInt;
      ReversalRetryPauseTimeMS : DInt;
      ReversalWindowTimer { S7_SetPoint := 'True'} : TON_TIME;
      ReversalStepEdge : Bool;
      ReversalStepEdgeMem : Bool;
      ReversalCount : Int;   // Reversals since the window last re-armed (not per-cycle, unlike the pusher's own PressureTripCount) - ReversalWindowTimer restarts the window every time this is above zero, so ReversalCountThreshold reversals must occur within one ReversalWindowTime of each other to raise ShredderBlockedFault, not just ReversalCountThreshold times ever.
      PreStartTimer { S7_SetPoint := 'True'} : TON_TIME;
      DischargeStartTimer { S7_SetPoint := 'True'} : TON_TIME;
      ReverseRunTimer { S7_SetPoint := 'True'} : TON_TIME;
      InfeedRestartTimer { S7_SetPoint := 'True'} : TON_TIME;
      UpstreamEnableTimer { S7_SetPoint := 'True'} : TON_TIME;
      InfeedRunning : Bool;   // Latched once InfeedRestartTimer has timed out from the last hopper-clear - drives RunInfeedConv directly and (after a further UpstreamEnableTimer delay) EnableUpstream.
      SpinUpTimer { S7_SetPoint := 'True'} : TON_TIME;
      OvercurrentMediumTimer { S7_SetPoint := 'True'} : TON_TIME;
      OvercurrentHighTimer { S7_SetPoint := 'True'} : TON_TIME;
      OvercurrentTripped : Bool;   // KNOWN GAP, not wired to real current yet: both timers below are gated 'AND NOT AlwaysTrue' (permanently false placeholders) because DB_AnalogInput.ShredderMotorCurrent > DB_Settings.OvercurrentSetpointMedium/High is a genuine Real-vs-Real comparison this converter's synthesizer can't type correctly yet (hardcodes Int) - flagged and deferred rather than guessed at. This bit, and Step 50's own overcurrent-abort transition, are dead code until that's built.
      OvercurrentAbortPauseTimer { S7_SetPoint := 'True'} : TON_TIME;
   END_VAR
   VAR_TEMP
      "Time" : Real;
   END_VAR
BEGIN

REGION Network 1: Stop Command
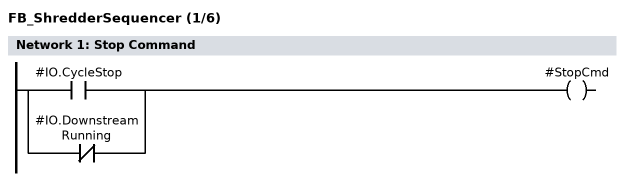
   RUNG wire#powerrail
      Contact( #IO.CycleStop )
      wire#w1
      Coil( #StopCmd )
   END_RUNG
   RUNG wire#powerrail
      I_Contact( #IO.DownstreamRunning )
   END_RUNG wire#w1
   // the same network as SCL:
   #StopCmd := #IO.CycleStop OR NOT #IO.DownstreamRunning;
END_REGION

REGION Network 2: HMI Time Conversions
   // HMI/DB_Settings times are Real seconds for operator legibility; every TON below needs its PT in DInt ms - one MUL+CONVERT pair per timer, matching the MotorDOL FTTime/EnableUPSTime idiom. Kept as one block up front rather than repeated at each timer, so the x1000 idiom is visibly consistent and only ever done once.
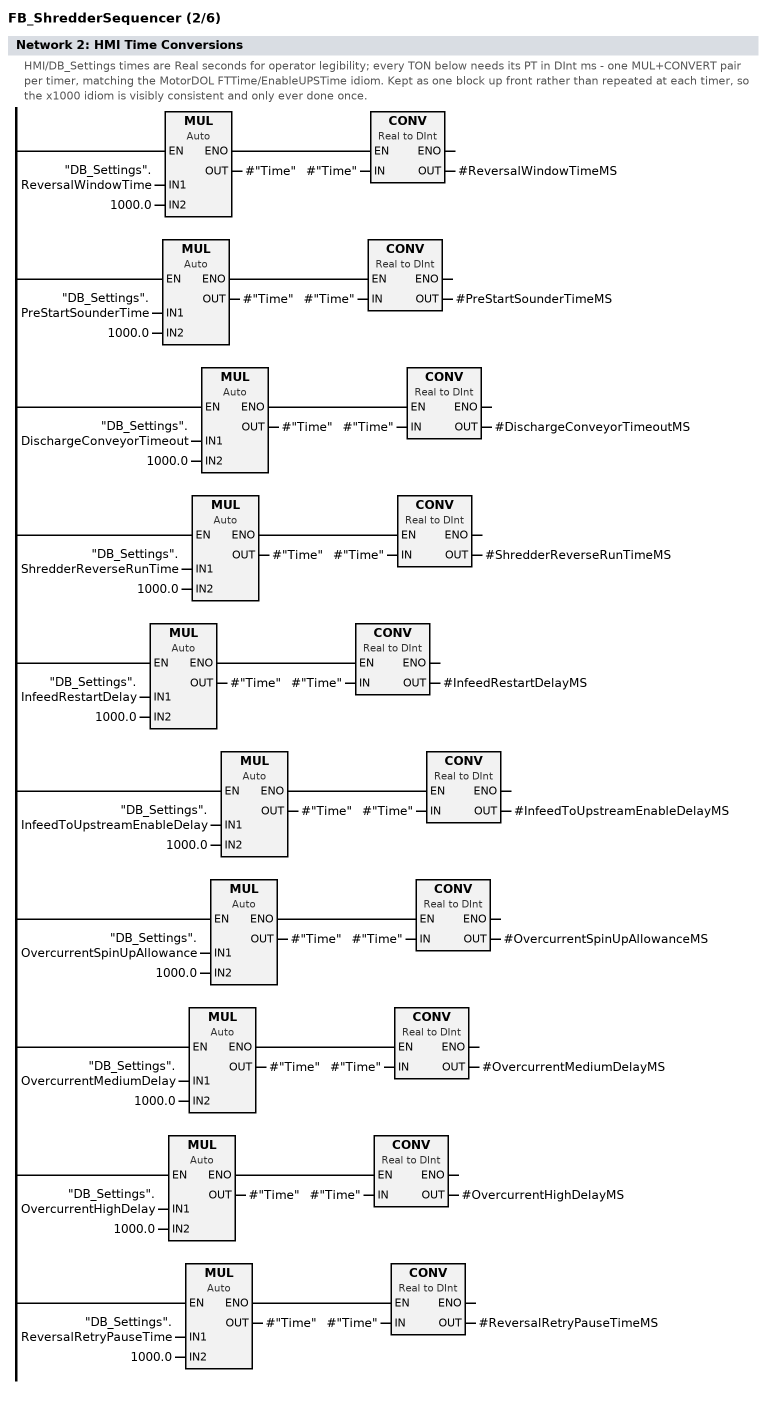
   RUNG wire#powerrail
      Mul(in1 := "DB_Settings".ReversalWindowTime, in2 := 1000.0, out => #"Time")
      { S7_Templates := "[SrcType := Real, DestType := DInt]" } Convert(in := #"Time", out => #ReversalWindowTimeMS)
   END_RUNG
   RUNG wire#powerrail
      Mul(in1 := "DB_Settings".PreStartSounderTime, in2 := 1000.0, out => #"Time")
      { S7_Templates := "[SrcType := Real, DestType := DInt]" } Convert(in := #"Time", out => #PreStartSounderTimeMS)
   END_RUNG
   RUNG wire#powerrail
      Mul(in1 := "DB_Settings".DischargeConveyorTimeout, in2 := 1000.0, out => #"Time")
      { S7_Templates := "[SrcType := Real, DestType := DInt]" } Convert(in := #"Time", out => #DischargeConveyorTimeoutMS)
   END_RUNG
   RUNG wire#powerrail
      Mul(in1 := "DB_Settings".ShredderReverseRunTime, in2 := 1000.0, out => #"Time")
      { S7_Templates := "[SrcType := Real, DestType := DInt]" } Convert(in := #"Time", out => #ShredderReverseRunTimeMS)
   END_RUNG
   RUNG wire#powerrail
      Mul(in1 := "DB_Settings".InfeedRestartDelay, in2 := 1000.0, out => #"Time")
      { S7_Templates := "[SrcType := Real, DestType := DInt]" } Convert(in := #"Time", out => #InfeedRestartDelayMS)
   END_RUNG
   RUNG wire#powerrail
      Mul(in1 := "DB_Settings".InfeedToUpstreamEnableDelay, in2 := 1000.0, out => #"Time")
      { S7_Templates := "[SrcType := Real, DestType := DInt]" } Convert(in := #"Time", out => #InfeedToUpstreamEnableDelayMS)
   END_RUNG
   RUNG wire#powerrail
      Mul(in1 := "DB_Settings".OvercurrentSpinUpAllowance, in2 := 1000.0, out => #"Time")
      { S7_Templates := "[SrcType := Real, DestType := DInt]" } Convert(in := #"Time", out => #OvercurrentSpinUpAllowanceMS)
   END_RUNG
   RUNG wire#powerrail
      Mul(in1 := "DB_Settings".OvercurrentMediumDelay, in2 := 1000.0, out => #"Time")
      { S7_Templates := "[SrcType := Real, DestType := DInt]" } Convert(in := #"Time", out => #OvercurrentMediumDelayMS)
   END_RUNG
   RUNG wire#powerrail
      Mul(in1 := "DB_Settings".OvercurrentHighDelay, in2 := 1000.0, out => #"Time")
      { S7_Templates := "[SrcType := Real, DestType := DInt]" } Convert(in := #"Time", out => #OvercurrentHighDelayMS)
   END_RUNG
   RUNG wire#powerrail
      Mul(in1 := "DB_Settings".ReversalRetryPauseTime, in2 := 1000.0, out => #"Time")
      { S7_Templates := "[SrcType := Real, DestType := DInt]" } Convert(in := #"Time", out => #ReversalRetryPauseTimeMS)
   END_RUNG
   // the same network as SCL:
   #"Time" := "DB_Settings".ReversalWindowTime * 1000.0;
   #ReversalWindowTimeMS := REAL_TO_DINT(#"Time");
   #"Time" := "DB_Settings".PreStartSounderTime * 1000.0;
   #PreStartSounderTimeMS := REAL_TO_DINT(#"Time");
   #"Time" := "DB_Settings".DischargeConveyorTimeout * 1000.0;
   #DischargeConveyorTimeoutMS := REAL_TO_DINT(#"Time");
   #"Time" := "DB_Settings".ShredderReverseRunTime * 1000.0;
   #ShredderReverseRunTimeMS := REAL_TO_DINT(#"Time");
   #"Time" := "DB_Settings".InfeedRestartDelay * 1000.0;
   #InfeedRestartDelayMS := REAL_TO_DINT(#"Time");
   #"Time" := "DB_Settings".InfeedToUpstreamEnableDelay * 1000.0;
   #InfeedToUpstreamEnableDelayMS := REAL_TO_DINT(#"Time");
   #"Time" := "DB_Settings".OvercurrentSpinUpAllowance * 1000.0;
   #OvercurrentSpinUpAllowanceMS := REAL_TO_DINT(#"Time");
   #"Time" := "DB_Settings".OvercurrentMediumDelay * 1000.0;
   #OvercurrentMediumDelayMS := REAL_TO_DINT(#"Time");
   #"Time" := "DB_Settings".OvercurrentHighDelay * 1000.0;
   #OvercurrentHighDelayMS := REAL_TO_DINT(#"Time");
   #"Time" := "DB_Settings".ReversalRetryPauseTime * 1000.0;
   #ReversalRetryPauseTimeMS := REAL_TO_DINT(#"Time");
END_REGION

REGION Network 3: Reversal Re-Arm Window Timer
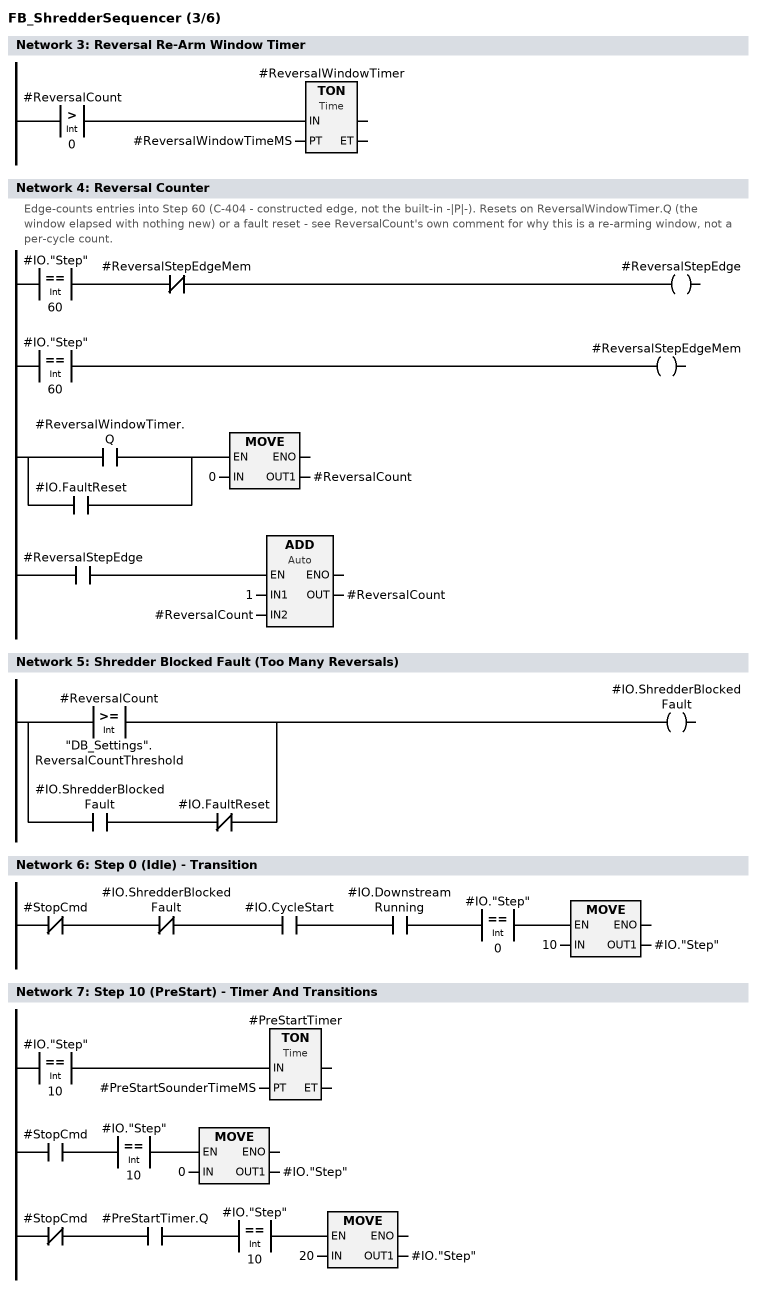
   RUNG wire#powerrail
      { S7_Templates := "SrcType := Int" } GT_Contact(in1 := #ReversalCount, in2 := 0)
      { S7_Templates := "time_type := Time" } #ReversalWindowTimer.TON(pt := #ReversalWindowTimeMS, et =>)
   END_RUNG
   // the same network as SCL:
   #ReversalWindowTimer(IN := #ReversalCount > 0, PT := #ReversalWindowTimeMS);   // TON
END_REGION

REGION Network 4: Reversal Counter
   // Edge-counts entries into Step 60 (C-404 - constructed edge, not the built-in -|P|-). Resets on ReversalWindowTimer.Q (the window elapsed with nothing new) or a fault reset - see ReversalCount's own comment for why this is a re-arming window, not a per-cycle count.
   RUNG wire#powerrail
      { S7_Templates := "SrcType := Int" } EQ_Contact(in1 := #IO."Step", in2 := 60)
      I_Contact( #ReversalStepEdgeMem )
      Coil( #ReversalStepEdge )
   END_RUNG
   RUNG wire#powerrail
      { S7_Templates := "SrcType := Int" } EQ_Contact(in1 := #IO."Step", in2 := 60)
      Coil( #ReversalStepEdgeMem )
   END_RUNG
   RUNG wire#powerrail
      Contact( #ReversalWindowTimer.Q )
      wire#w1
      Move(in := 0, out1 => #ReversalCount)
   END_RUNG
   RUNG wire#powerrail
      Contact( #IO.FaultReset )
   END_RUNG wire#w1
   RUNG wire#powerrail
      Contact( #ReversalStepEdge )
      Add(in1 := 1, in2 := #ReversalCount, out => #ReversalCount)
   END_RUNG
   // the same network as SCL:
   #ReversalStepEdge := (#IO."Step" = 60) AND NOT #ReversalStepEdgeMem;
   #ReversalStepEdgeMem := #IO."Step" = 60;
   IF #ReversalWindowTimer.Q OR #IO.FaultReset THEN #ReversalCount := 0; END_IF;
   IF #ReversalStepEdge THEN #ReversalCount := 1 + #ReversalCount; END_IF;
END_REGION

REGION Network 5: Shredder Blocked Fault (Too Many Reversals)
   RUNG wire#powerrail
      { S7_Templates := "SrcType := Int" } GE_Contact(in1 := #ReversalCount, in2 := "DB_Settings".ReversalCountThreshold)
      wire#w1
      Coil( #IO.ShredderBlockedFault )
   END_RUNG
   RUNG wire#powerrail
      Contact( #IO.ShredderBlockedFault )
      I_Contact( #IO.FaultReset )
   END_RUNG wire#w1
   // the same network as SCL:
   #IO.ShredderBlockedFault := (#ReversalCount >= "DB_Settings".ReversalCountThreshold) OR (#IO.ShredderBlockedFault AND NOT #IO.FaultReset);
END_REGION

REGION Network 6: Step 0 (Idle) - Transition
   RUNG wire#powerrail
      I_Contact( #StopCmd )
      I_Contact( #IO.ShredderBlockedFault )
      Contact( #IO.CycleStart )
      Contact( #IO.DownstreamRunning )
      { S7_Templates := "SrcType := Int" } EQ_Contact(in1 := #IO."Step", in2 := 0)
      Move(in := 10, out1 => #IO."Step")
   END_RUNG
   // the same network as SCL:
   IF NOT #StopCmd AND NOT #IO.ShredderBlockedFault AND #IO.CycleStart AND #IO.DownstreamRunning AND (#IO."Step" = 0) THEN
       #IO."Step" := 10;
   END_IF;
END_REGION

REGION Network 7: Step 10 (PreStart) - Timer And Transitions
   RUNG wire#powerrail
      { S7_Templates := "SrcType := Int" } EQ_Contact(in1 := #IO."Step", in2 := 10)
      { S7_Templates := "time_type := Time" } #PreStartTimer.TON(pt := #PreStartSounderTimeMS, et =>)
   END_RUNG
   RUNG wire#powerrail
      Contact( #StopCmd )
      { S7_Templates := "SrcType := Int" } EQ_Contact(in1 := #IO."Step", in2 := 10)
      Move(in := 0, out1 => #IO."Step")
   END_RUNG
   RUNG wire#powerrail
      I_Contact( #StopCmd )
      Contact( #PreStartTimer.Q )
      { S7_Templates := "SrcType := Int" } EQ_Contact(in1 := #IO."Step", in2 := 10)
      Move(in := 20, out1 => #IO."Step")
   END_RUNG
   // the same network as SCL:
   #PreStartTimer(IN := #IO."Step" = 10, PT := #PreStartSounderTimeMS);   // TON
   IF #StopCmd AND (#IO."Step" = 10) THEN #IO."Step" := 0; END_IF;
   IF NOT #StopCmd AND #PreStartTimer.Q AND (#IO."Step" = 10) THEN #IO."Step" := 20; END_IF;
END_REGION

REGION Network 8: Step 20 (DischargeStart) - Timer, Timeout Fault, And Transitions
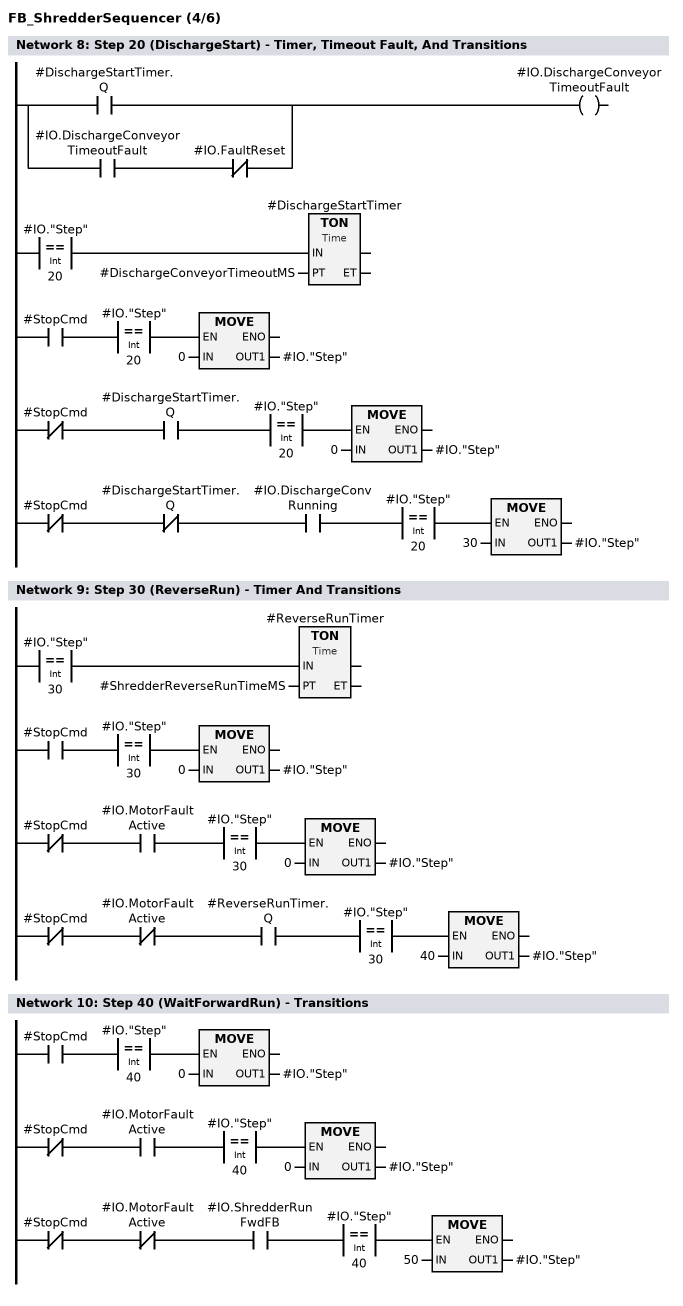
   RUNG wire#powerrail
      Contact( #DischargeStartTimer.Q )
      wire#w1
      Coil( #IO.DischargeConveyorTimeoutFault )
   END_RUNG
   RUNG wire#powerrail
      Contact( #IO.DischargeConveyorTimeoutFault )
      I_Contact( #IO.FaultReset )
   END_RUNG wire#w1
   RUNG wire#powerrail
      { S7_Templates := "SrcType := Int" } EQ_Contact(in1 := #IO."Step", in2 := 20)
      { S7_Templates := "time_type := Time" } #DischargeStartTimer.TON(pt := #DischargeConveyorTimeoutMS, et =>)
   END_RUNG
   RUNG wire#powerrail
      Contact( #StopCmd )
      { S7_Templates := "SrcType := Int" } EQ_Contact(in1 := #IO."Step", in2 := 20)
      Move(in := 0, out1 => #IO."Step")
   END_RUNG
   RUNG wire#powerrail
      I_Contact( #StopCmd )
      Contact( #DischargeStartTimer.Q )
      { S7_Templates := "SrcType := Int" } EQ_Contact(in1 := #IO."Step", in2 := 20)
      Move(in := 0, out1 => #IO."Step")
   END_RUNG
   RUNG wire#powerrail
      I_Contact( #StopCmd )
      I_Contact( #DischargeStartTimer.Q )
      Contact( #IO.DischargeConvRunning )
      { S7_Templates := "SrcType := Int" } EQ_Contact(in1 := #IO."Step", in2 := 20)
      Move(in := 30, out1 => #IO."Step")
   END_RUNG
   // the same network as SCL:
   #IO.DischargeConveyorTimeoutFault := #DischargeStartTimer.Q OR (#IO.DischargeConveyorTimeoutFault AND NOT #IO.FaultReset);
   #DischargeStartTimer(IN := #IO."Step" = 20, PT := #DischargeConveyorTimeoutMS);   // TON
   IF #StopCmd AND (#IO."Step" = 20) THEN #IO."Step" := 0; END_IF;
   IF NOT #StopCmd AND #DischargeStartTimer.Q AND (#IO."Step" = 20) THEN #IO."Step" := 0; END_IF;
   IF NOT #StopCmd AND NOT #DischargeStartTimer.Q AND #IO.DischargeConvRunning AND (#IO."Step" = 20) THEN
       #IO."Step" := 30;
   END_IF;
END_REGION

REGION Network 9: Step 30 (ReverseRun) - Timer And Transitions
   RUNG wire#powerrail
      { S7_Templates := "SrcType := Int" } EQ_Contact(in1 := #IO."Step", in2 := 30)
      { S7_Templates := "time_type := Time" } #ReverseRunTimer.TON(pt := #ShredderReverseRunTimeMS, et =>)
   END_RUNG
   RUNG wire#powerrail
      Contact( #StopCmd )
      { S7_Templates := "SrcType := Int" } EQ_Contact(in1 := #IO."Step", in2 := 30)
      Move(in := 0, out1 => #IO."Step")
   END_RUNG
   RUNG wire#powerrail
      I_Contact( #StopCmd )
      Contact( #IO.MotorFaultActive )
      { S7_Templates := "SrcType := Int" } EQ_Contact(in1 := #IO."Step", in2 := 30)
      Move(in := 0, out1 => #IO."Step")
   END_RUNG
   RUNG wire#powerrail
      I_Contact( #StopCmd )
      I_Contact( #IO.MotorFaultActive )
      Contact( #ReverseRunTimer.Q )
      { S7_Templates := "SrcType := Int" } EQ_Contact(in1 := #IO."Step", in2 := 30)
      Move(in := 40, out1 => #IO."Step")
   END_RUNG
   // the same network as SCL:
   #ReverseRunTimer(IN := #IO."Step" = 30, PT := #ShredderReverseRunTimeMS);   // TON
   IF #StopCmd AND (#IO."Step" = 30) THEN #IO."Step" := 0; END_IF;
   IF NOT #StopCmd AND #IO.MotorFaultActive AND (#IO."Step" = 30) THEN #IO."Step" := 0; END_IF;
   IF NOT #StopCmd AND NOT #IO.MotorFaultActive AND #ReverseRunTimer.Q AND (#IO."Step" = 30) THEN
       #IO."Step" := 40;
   END_IF;
END_REGION

REGION Network 10: Step 40 (WaitForwardRun) - Transitions
   RUNG wire#powerrail
      Contact( #StopCmd )
      { S7_Templates := "SrcType := Int" } EQ_Contact(in1 := #IO."Step", in2 := 40)
      Move(in := 0, out1 => #IO."Step")
   END_RUNG
   RUNG wire#powerrail
      I_Contact( #StopCmd )
      Contact( #IO.MotorFaultActive )
      { S7_Templates := "SrcType := Int" } EQ_Contact(in1 := #IO."Step", in2 := 40)
      Move(in := 0, out1 => #IO."Step")
   END_RUNG
   RUNG wire#powerrail
      I_Contact( #StopCmd )
      I_Contact( #IO.MotorFaultActive )
      Contact( #IO.ShredderRunFwdFB )
      { S7_Templates := "SrcType := Int" } EQ_Contact(in1 := #IO."Step", in2 := 40)
      Move(in := 50, out1 => #IO."Step")
   END_RUNG
   // the same network as SCL:
   IF #StopCmd AND (#IO."Step" = 40) THEN #IO."Step" := 0; END_IF;
   IF NOT #StopCmd AND #IO.MotorFaultActive AND (#IO."Step" = 40) THEN #IO."Step" := 0; END_IF;
   IF NOT #StopCmd AND NOT #IO.MotorFaultActive AND #IO.ShredderRunFwdFB AND (#IO."Step" = 40) THEN
       #IO."Step" := 50;
   END_IF;
END_REGION

REGION Network 11: Step 50 (Running) - Infeed Restart, Upstream Enable, And Outputs
   // UpstreamEnableTimer's own IN reads InfeedRunning one scan behind this network's own InfeedRunning update below (it's kind-ordered before the coil that writes it) - harmless for a multi-second delay, and matches this design's original timing exactly. EnableUpstream lives here, next to its own timer, rather than in the general Output Commands network - this is the output the MotorFwdRevSystem CALL-site correction was specifically about: it must only ever come from Step=50 dwell time, never from motor-running telemetry.
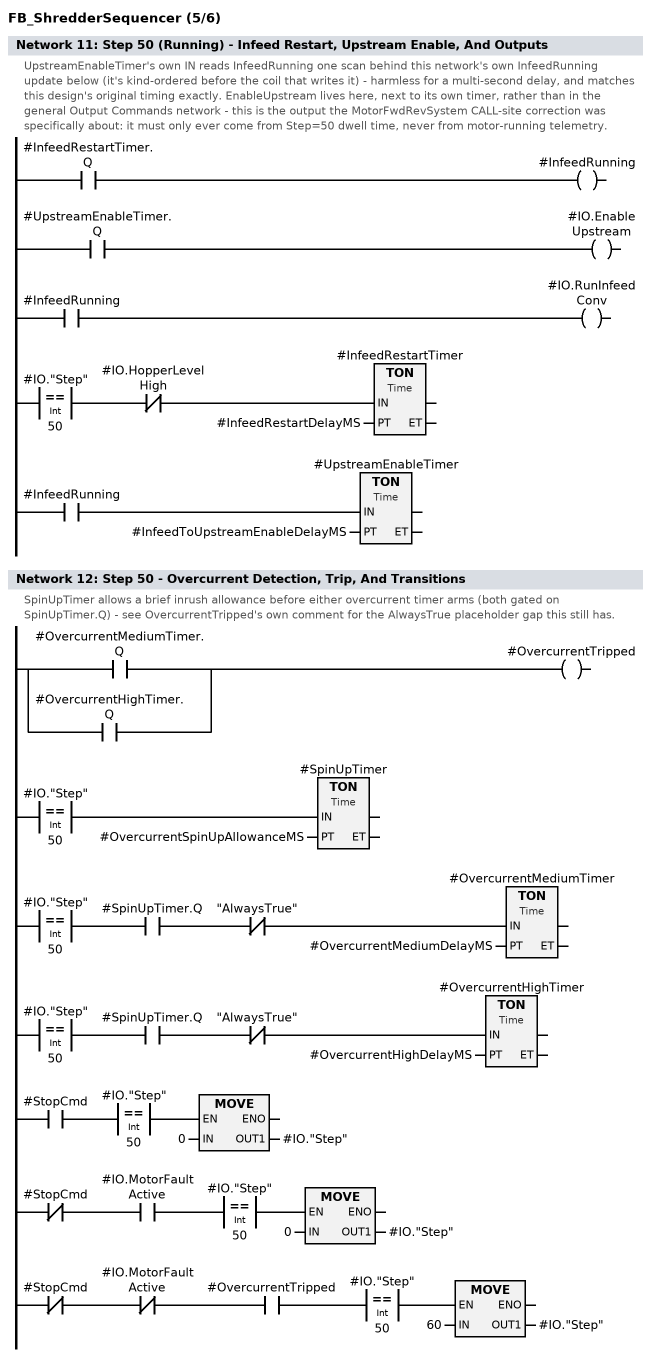
   RUNG wire#powerrail
      Contact( #InfeedRestartTimer.Q )
      Coil( #InfeedRunning )
   END_RUNG
   RUNG wire#powerrail
      Contact( #UpstreamEnableTimer.Q )
      Coil( #IO.EnableUpstream )
   END_RUNG
   RUNG wire#powerrail
      Contact( #InfeedRunning )
      Coil( #IO.RunInfeedConv )
   END_RUNG
   RUNG wire#powerrail
      { S7_Templates := "SrcType := Int" } EQ_Contact(in1 := #IO."Step", in2 := 50)
      I_Contact( #IO.HopperLevelHigh )
      { S7_Templates := "time_type := Time" } #InfeedRestartTimer.TON(pt := #InfeedRestartDelayMS, et =>)
   END_RUNG
   RUNG wire#powerrail
      Contact( #InfeedRunning )
      { S7_Templates := "time_type := Time" } #UpstreamEnableTimer.TON(pt := #InfeedToUpstreamEnableDelayMS, et =>)
   END_RUNG
   // the same network as SCL:
   #InfeedRunning := #InfeedRestartTimer.Q;
   #IO.EnableUpstream := #UpstreamEnableTimer.Q;
   #IO.RunInfeedConv := #InfeedRunning;
   #InfeedRestartTimer(IN := (#IO."Step" = 50) AND NOT #IO.HopperLevelHigh, PT := #InfeedRestartDelayMS);   // TON
   #UpstreamEnableTimer(IN := #InfeedRunning, PT := #InfeedToUpstreamEnableDelayMS);   // TON
END_REGION

REGION Network 12: Step 50 - Overcurrent Detection, Trip, And Transitions
   // SpinUpTimer allows a brief inrush allowance before either overcurrent timer arms (both gated on SpinUpTimer.Q) - see OvercurrentTripped's own comment for the AlwaysTrue placeholder gap this still has.
   RUNG wire#powerrail
      Contact( #OvercurrentMediumTimer.Q )
      wire#w1
      Coil( #OvercurrentTripped )
   END_RUNG
   RUNG wire#powerrail
      Contact( #OvercurrentHighTimer.Q )
   END_RUNG wire#w1
   RUNG wire#powerrail
      { S7_Templates := "SrcType := Int" } EQ_Contact(in1 := #IO."Step", in2 := 50)
      { S7_Templates := "time_type := Time" } #SpinUpTimer.TON(pt := #OvercurrentSpinUpAllowanceMS, et =>)
   END_RUNG
   RUNG wire#powerrail
      { S7_Templates := "SrcType := Int" } EQ_Contact(in1 := #IO."Step", in2 := 50)
      Contact( #SpinUpTimer.Q )
      I_Contact( "AlwaysTrue" )
      { S7_Templates := "time_type := Time" } #OvercurrentMediumTimer.TON(pt := #OvercurrentMediumDelayMS, et =>)
   END_RUNG
   RUNG wire#powerrail
      { S7_Templates := "SrcType := Int" } EQ_Contact(in1 := #IO."Step", in2 := 50)
      Contact( #SpinUpTimer.Q )
      I_Contact( "AlwaysTrue" )
      { S7_Templates := "time_type := Time" } #OvercurrentHighTimer.TON(pt := #OvercurrentHighDelayMS, et =>)
   END_RUNG
   RUNG wire#powerrail
      Contact( #StopCmd )
      { S7_Templates := "SrcType := Int" } EQ_Contact(in1 := #IO."Step", in2 := 50)
      Move(in := 0, out1 => #IO."Step")
   END_RUNG
   RUNG wire#powerrail
      I_Contact( #StopCmd )
      Contact( #IO.MotorFaultActive )
      { S7_Templates := "SrcType := Int" } EQ_Contact(in1 := #IO."Step", in2 := 50)
      Move(in := 0, out1 => #IO."Step")
   END_RUNG
   RUNG wire#powerrail
      I_Contact( #StopCmd )
      I_Contact( #IO.MotorFaultActive )
      Contact( #OvercurrentTripped )
      { S7_Templates := "SrcType := Int" } EQ_Contact(in1 := #IO."Step", in2 := 50)
      Move(in := 60, out1 => #IO."Step")
   END_RUNG
   // the same network as SCL:
   #OvercurrentTripped := #OvercurrentMediumTimer.Q OR #OvercurrentHighTimer.Q;
   #SpinUpTimer(IN := #IO."Step" = 50, PT := #OvercurrentSpinUpAllowanceMS);   // TON
   #OvercurrentMediumTimer(IN := (#IO."Step" = 50) AND #SpinUpTimer.Q AND NOT "AlwaysTrue",   // TON
                           PT := #OvercurrentMediumDelayMS);
   #OvercurrentHighTimer(IN := (#IO."Step" = 50) AND #SpinUpTimer.Q AND NOT "AlwaysTrue",   // TON
                         PT := #OvercurrentHighDelayMS);
   IF #StopCmd AND (#IO."Step" = 50) THEN #IO."Step" := 0; END_IF;
   IF NOT #StopCmd AND #IO.MotorFaultActive AND (#IO."Step" = 50) THEN #IO."Step" := 0; END_IF;
   IF NOT #StopCmd AND NOT #IO.MotorFaultActive AND #OvercurrentTripped AND (#IO."Step" = 50) THEN
       #IO."Step" := 60;
   END_IF;
END_REGION

REGION Network 13: Step 60 (OvercurrentAbort) - Timer And Transitions
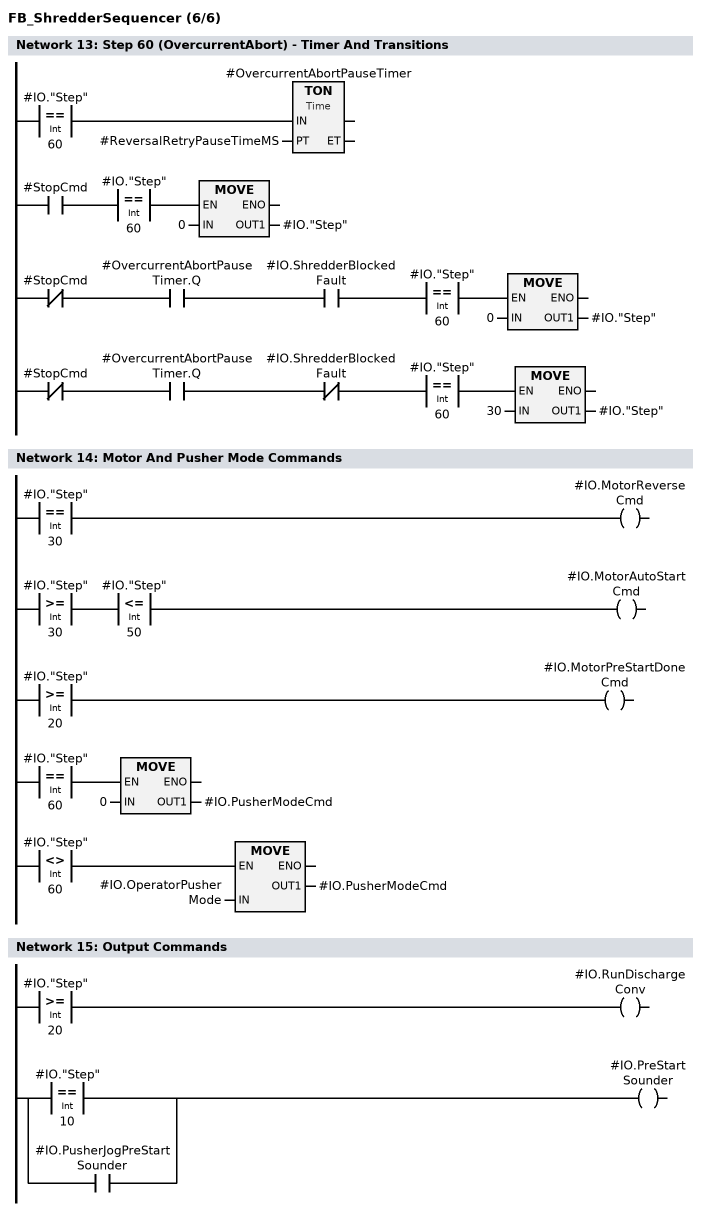
   RUNG wire#powerrail
      { S7_Templates := "SrcType := Int" } EQ_Contact(in1 := #IO."Step", in2 := 60)
      { S7_Templates := "time_type := Time" } #OvercurrentAbortPauseTimer.TON(pt := #ReversalRetryPauseTimeMS, et =>)
   END_RUNG
   RUNG wire#powerrail
      Contact( #StopCmd )
      { S7_Templates := "SrcType := Int" } EQ_Contact(in1 := #IO."Step", in2 := 60)
      Move(in := 0, out1 => #IO."Step")
   END_RUNG
   RUNG wire#powerrail
      I_Contact( #StopCmd )
      Contact( #OvercurrentAbortPauseTimer.Q )
      Contact( #IO.ShredderBlockedFault )
      { S7_Templates := "SrcType := Int" } EQ_Contact(in1 := #IO."Step", in2 := 60)
      Move(in := 0, out1 => #IO."Step")
   END_RUNG
   RUNG wire#powerrail
      I_Contact( #StopCmd )
      Contact( #OvercurrentAbortPauseTimer.Q )
      I_Contact( #IO.ShredderBlockedFault )
      { S7_Templates := "SrcType := Int" } EQ_Contact(in1 := #IO."Step", in2 := 60)
      Move(in := 30, out1 => #IO."Step")
   END_RUNG
   // the same network as SCL:
   #OvercurrentAbortPauseTimer(IN := #IO."Step" = 60, PT := #ReversalRetryPauseTimeMS);   // TON
   IF #StopCmd AND (#IO."Step" = 60) THEN #IO."Step" := 0; END_IF;
   IF NOT #StopCmd AND #OvercurrentAbortPauseTimer.Q AND #IO.ShredderBlockedFault AND (#IO."Step" = 60) THEN
       #IO."Step" := 0;
   END_IF;
   IF NOT #StopCmd AND #OvercurrentAbortPauseTimer.Q AND NOT #IO.ShredderBlockedFault AND (#IO."Step" = 60) THEN
       #IO."Step" := 30;
   END_IF;
END_REGION

REGION Network 14: Motor And Pusher Mode Commands
   RUNG wire#powerrail
      { S7_Templates := "SrcType := Int" } EQ_Contact(in1 := #IO."Step", in2 := 30)
      Coil( #IO.MotorReverseCmd )
   END_RUNG
   RUNG wire#powerrail
      { S7_Templates := "SrcType := Int" } GE_Contact(in1 := #IO."Step", in2 := 30)
      { S7_Templates := "SrcType := Int" } LE_Contact(in1 := #IO."Step", in2 := 50)
      Coil( #IO.MotorAutoStartCmd )
   END_RUNG
   RUNG wire#powerrail
      { S7_Templates := "SrcType := Int" } GE_Contact(in1 := #IO."Step", in2 := 20)
      Coil( #IO.MotorPreStartDoneCmd )
   END_RUNG
   RUNG wire#powerrail
      { S7_Templates := "SrcType := Int" } EQ_Contact(in1 := #IO."Step", in2 := 60)
      Move(in := 0, out1 => #IO.PusherModeCmd)
   END_RUNG
   RUNG wire#powerrail
      { S7_Templates := "SrcType := Int" } NE_Contact(in1 := #IO."Step", in2 := 60)
      Move(in := #IO.OperatorPusherMode, out1 => #IO.PusherModeCmd)
   END_RUNG
   // the same network as SCL:
   #IO.MotorReverseCmd := #IO."Step" = 30;
   #IO.MotorAutoStartCmd := (#IO."Step" >= 30) AND (#IO."Step" <= 50);
   #IO.MotorPreStartDoneCmd := #IO."Step" >= 20;
   IF #IO."Step" = 60 THEN #IO.PusherModeCmd := 0; END_IF;
   IF #IO."Step" <> 60 THEN #IO.PusherModeCmd := #IO.OperatorPusherMode; END_IF;
END_REGION

REGION Network 15: Output Commands
   RUNG wire#powerrail
      { S7_Templates := "SrcType := Int" } GE_Contact(in1 := #IO."Step", in2 := 20)
      Coil( #IO.RunDischargeConv )
   END_RUNG
   RUNG wire#powerrail
      { S7_Templates := "SrcType := Int" } EQ_Contact(in1 := #IO."Step", in2 := 10)
      wire#w1
      Coil( #IO.PreStartSounder )
   END_RUNG
   RUNG wire#powerrail
      Contact( #IO.PusherJogPreStartSounder )
   END_RUNG wire#w1
   // the same network as SCL:
   #IO.RunDischargeConv := #IO."Step" >= 20;
   #IO.PreStartSounder := (#IO."Step" = 10) OR #IO.PusherJogPreStartSounder;
END_REGION
END_FUNCTION_BLOCK

FUNCTION_BLOCK "FB_MotorFwdRevSystem"   // FB7, LAD
{ S7_Optimized_Access := 'TRUE' }
VERSION : 0.1
// stored: AutoNumber true, IsIECCheckEnabled false, IsRetainMemResEnabled false, MemoryReserve 100, SetENOAutomatically false, UDAEnableTagReadback false
   VAR RETAIN
      IO : "MotorFwdRevIOSet";
   END_VAR
   VAR
      RisingEdgeFlags : Array[0..3] of Bool;
      NegitiveSignalEdge : Array[0..2] of Bool;
      Pasue : Bool;
      HrTotaliserTimerReset : Bool;
      EnableUPSTimeMS : DInt;
      ShutdownTimeMS : DInt;
      FTTimeMS : DInt;
      PauseTimeMS : DInt;
      ReverseIgnoreFTTimeMS : DInt;
      FaultTripTimer { S7_SetPoint := 'True'} : TON_TIME;
      FTSTimer { S7_SetPoint := 'True'} : TON_TIME;
      EnableUpstreamTimer { S7_SetPoint := 'True'} : TON_TIME;
      ShutdownTimer { S7_SetPoint := 'True'} : TON_TIME;
      GeneralDelayTimer { S7_SetPoint := 'True'} : TON_TIME;
      InHandReqPreStart { S7_SetPoint := 'True'} : TON_TIME;
      CycleDelayReset { S7_SetPoint := 'True'} : TON_TIME;
   END_VAR
   VAR RETAIN
      HrTotaliserTimer { S7_SetPoint := 'True'} : TONR_TIME;
   END_VAR
   VAR
      ReversalPauseTimer { S7_SetPoint := 'True'} : TON_TIME;
      ReversalIgnoreFTTimer { S7_SetPoint := 'True'} : TON_TIME;
      PreStartMemory { S7_SetPoint := 'True'} : Bool;
      HandPosEdge : Bool;
      HandNegEdge : Bool;
      CycleDelay : Bool;
   END_VAR
   VAR_TEMP
      "Time" : Real;
      StartTimer : Bool;
   END_VAR
   VAR_TEMP   // added for the SCL form of the ladder/FBD networks
      _w1 : Bool;
      _w2 : Bool;
   END_VAR
BEGIN

REGION Network 1: Reverse Pause and Control
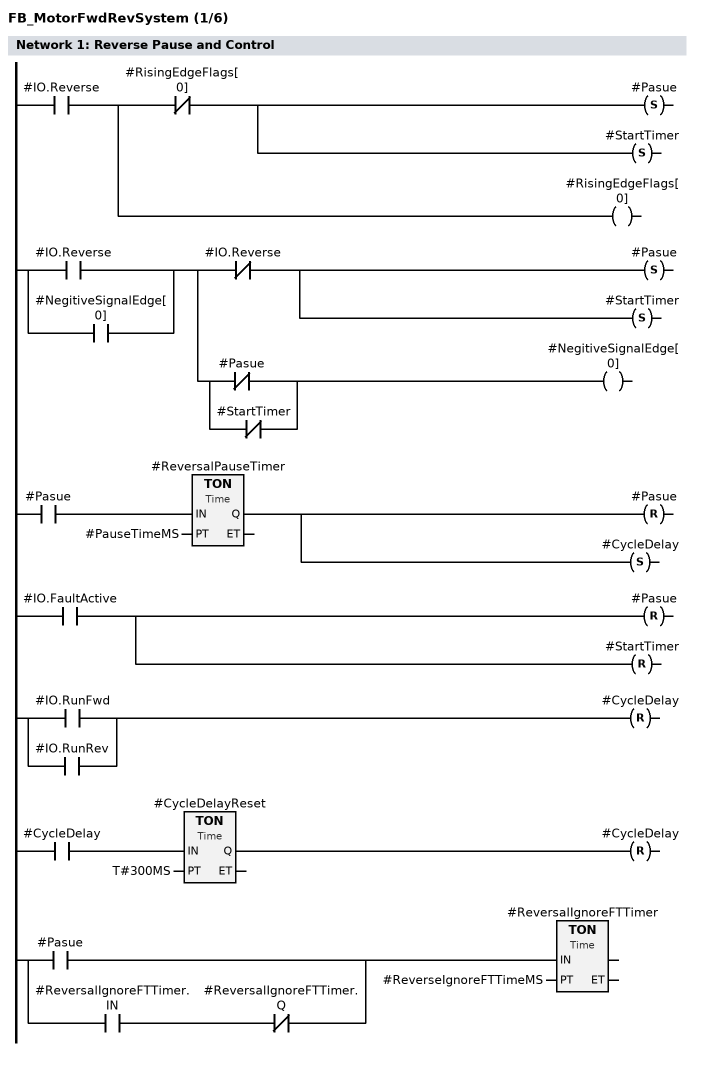
   RUNG wire#powerrail
      Contact( #IO.Reverse )
      wire#w1
      I_Contact( #RisingEdgeFlags[0] )
      wire#w2
      S_Coil( #Pasue )
   END_RUNG
   RUNG wire#w2
      S_Coil( #StartTimer )
   END_RUNG
   RUNG wire#w1
      Coil( #RisingEdgeFlags[0] )
   END_RUNG
   RUNG wire#powerrail
      Contact( #IO.Reverse )
      wire#w3
      I_Contact( #IO.Reverse )
      wire#w4
      S_Coil( #Pasue )
   END_RUNG
   RUNG wire#powerrail
      Contact( #NegitiveSignalEdge[0] )
   END_RUNG wire#w3
   RUNG wire#w4
      S_Coil( #StartTimer )
   END_RUNG
   RUNG wire#w3
      I_Contact( #Pasue )
      wire#w5
      Coil( #NegitiveSignalEdge[0] )
   END_RUNG
   RUNG wire#w3
      I_Contact( #StartTimer )
   END_RUNG wire#w5
   RUNG wire#powerrail
      Contact( #Pasue )
      { S7_Templates := "time_type := Time" } #ReversalPauseTimer.TON(pt := #PauseTimeMS, et =>)
      wire#w6
      R_Coil( #Pasue )
   END_RUNG
   RUNG wire#w6
      S_Coil( #CycleDelay )
   END_RUNG
   RUNG wire#powerrail
      Contact( #IO.FaultActive )
      wire#w7
      R_Coil( #Pasue )
   END_RUNG
   RUNG wire#w7
      R_Coil( #StartTimer )
   END_RUNG
   RUNG wire#powerrail
      Contact( #IO.RunFwd )
      wire#w8
      R_Coil( #CycleDelay )
   END_RUNG
   RUNG wire#powerrail
      Contact( #IO.RunRev )
   END_RUNG wire#w8
   RUNG wire#powerrail
      Contact( #CycleDelay )
      { S7_Templates := "time_type := Time" } #CycleDelayReset.TON(pt := T#300MS, et =>)
      R_Coil( #CycleDelay )
   END_RUNG
   RUNG wire#powerrail
      Contact( #Pasue )
      wire#w9
      { S7_Templates := "time_type := Time" } #ReversalIgnoreFTTimer.TON(pt := #ReverseIgnoreFTTimeMS, et =>)
   END_RUNG
   RUNG wire#powerrail
      Contact( #ReversalIgnoreFTTimer.IN )
      I_Contact( #ReversalIgnoreFTTimer.Q )
   END_RUNG wire#w9
   // the same network as SCL:
   IF #IO.Reverse AND NOT #RisingEdgeFlags[0] THEN
       #Pasue := TRUE;
       #StartTimer := TRUE;
   END_IF;
   #RisingEdgeFlags[0] := #IO.Reverse;
   #_w1 := #IO.Reverse OR #NegitiveSignalEdge[0];
   IF #_w1 AND NOT #IO.Reverse THEN
       #Pasue := TRUE;
       #StartTimer := TRUE;
   END_IF;
   #NegitiveSignalEdge[0] := #_w1 AND (NOT #Pasue OR NOT #StartTimer);
   #ReversalPauseTimer(IN := #Pasue, PT := #PauseTimeMS);   // TON
   IF #ReversalPauseTimer.Q THEN
       #Pasue := FALSE;
       #CycleDelay := TRUE;
   END_IF;
   IF #IO.FaultActive THEN
       #Pasue := FALSE;
       #StartTimer := FALSE;
   END_IF;
   IF #IO.RunFwd OR #IO.RunRev THEN #CycleDelay := FALSE; END_IF;
   #CycleDelayReset(IN := #CycleDelay, PT := T#300MS);   // TON
   IF #CycleDelayReset.Q THEN #CycleDelay := FALSE; END_IF;
   #ReversalIgnoreFTTimer(IN := #Pasue OR (#ReversalIgnoreFTTimer.IN AND NOT #ReversalIgnoreFTTimer.Q),   // TON
                          PT := #ReverseIgnoreFTTimeMS);
END_REGION

REGION Network 2: DOL Motor Start / Stop
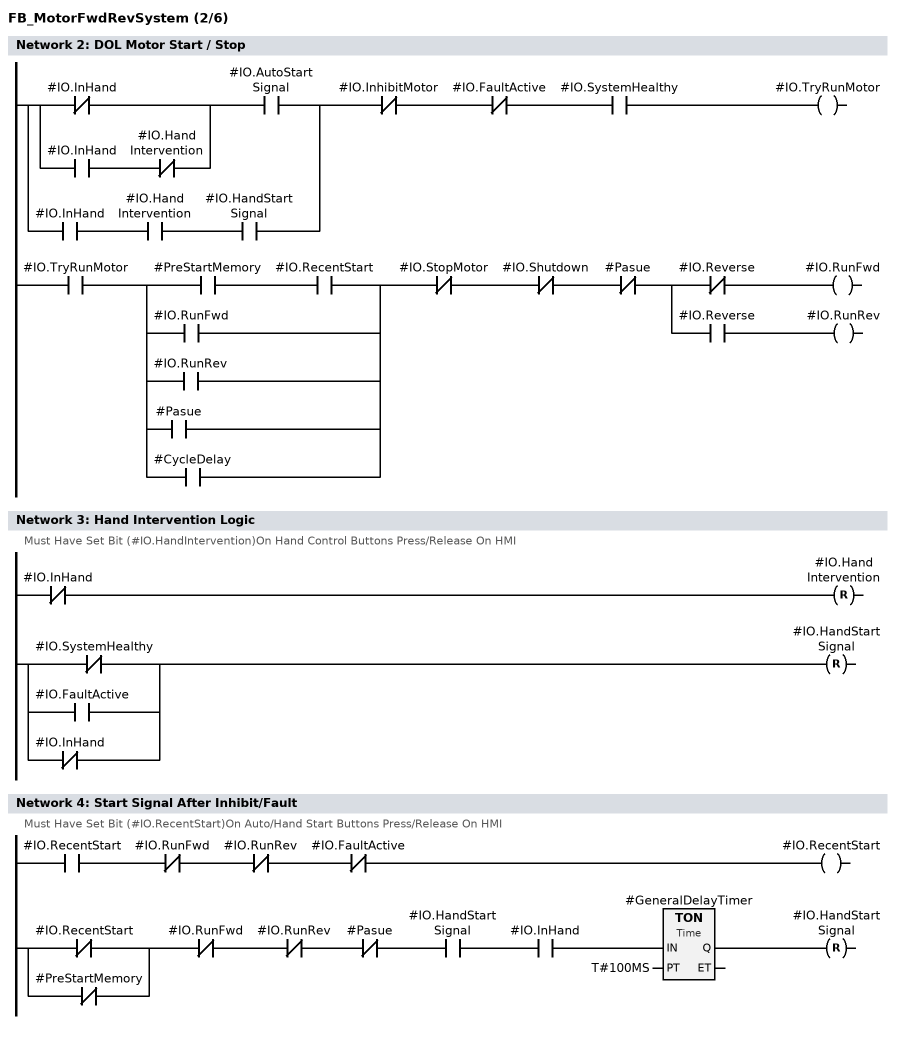
   RUNG wire#powerrail
      I_Contact( #IO.InHand )
      wire#w1
      Contact( #IO.AutoStartSignal )
      wire#w2
      I_Contact( #IO.InhibitMotor )
      I_Contact( #IO.FaultActive )
      Contact( #IO.SystemHealthy )
      Coil( #IO.TryRunMotor )
   END_RUNG
   RUNG wire#powerrail
      Contact( #IO.InHand )
      I_Contact( #IO.HandIntervention )
   END_RUNG wire#w1
   RUNG wire#powerrail
      Contact( #IO.InHand )
      Contact( #IO.HandIntervention )
      Contact( #IO.HandStartSignal )
   END_RUNG wire#w2
   RUNG wire#powerrail
      Contact( #IO.TryRunMotor )
      wire#w3
      Contact( #PreStartMemory )
      Contact( #IO.RecentStart )
      wire#w4
      I_Contact( #IO.StopMotor )
      I_Contact( #IO.Shutdown )
      I_Contact( #Pasue )
      wire#w5
      I_Contact( #IO.Reverse )
      Coil( #IO.RunFwd )
   END_RUNG
   RUNG wire#w3
      Contact( #IO.RunFwd )
   END_RUNG wire#w4
   RUNG wire#w3
      Contact( #IO.RunRev )
   END_RUNG wire#w4
   RUNG wire#w3
      Contact( #Pasue )
   END_RUNG wire#w4
   RUNG wire#w3
      Contact( #CycleDelay )
   END_RUNG wire#w4
   RUNG wire#w5
      Contact( #IO.Reverse )
      Coil( #IO.RunRev )
   END_RUNG
   // the same network as SCL:
   #IO.TryRunMotor := (((NOT #IO.InHand OR (#IO.InHand AND NOT #IO.HandIntervention)) AND #IO.AutoStartSignal) OR (#IO.InHand AND #IO.HandIntervention AND #IO.HandStartSignal)) AND NOT #IO.InhibitMotor AND NOT #IO.FaultActive AND #IO.SystemHealthy;
   #_w1 := #IO.TryRunMotor AND ((#PreStartMemory AND #IO.RecentStart) OR #IO.RunFwd OR #IO.RunRev OR #Pasue OR #CycleDelay) AND NOT #IO.StopMotor AND NOT #IO.Shutdown AND NOT #Pasue;
   #IO.RunFwd := #_w1 AND NOT #IO.Reverse;
   #IO.RunRev := #_w1 AND #IO.Reverse;
END_REGION

REGION Network 3: Hand Intervention Logic
   // Must Have Set Bit (#IO.HandIntervention)On Hand Control Buttons Press/Release On HMI
   RUNG wire#powerrail
      I_Contact( #IO.InHand )
      R_Coil( #IO.HandIntervention )
   END_RUNG
   RUNG wire#powerrail
      I_Contact( #IO.SystemHealthy )
      wire#w1
      R_Coil( #IO.HandStartSignal )
   END_RUNG
   RUNG wire#powerrail
      Contact( #IO.FaultActive )
   END_RUNG wire#w1
   RUNG wire#powerrail
      I_Contact( #IO.InHand )
   END_RUNG wire#w1
   // the same network as SCL:
   IF NOT #IO.InHand THEN #IO.HandIntervention := FALSE; END_IF;
   IF NOT #IO.SystemHealthy OR #IO.FaultActive OR NOT #IO.InHand THEN #IO.HandStartSignal := FALSE; END_IF;
END_REGION

REGION Network 4: Start Signal After Inhibit/Fault
   // Must Have Set Bit (#IO.RecentStart)On Auto/Hand Start Buttons Press/Release On HMI
   RUNG wire#powerrail
      Contact( #IO.RecentStart )
      I_Contact( #IO.RunFwd )
      I_Contact( #IO.RunRev )
      I_Contact( #IO.FaultActive )
      Coil( #IO.RecentStart )
   END_RUNG
   RUNG wire#powerrail
      I_Contact( #IO.RecentStart )
      wire#w1
      I_Contact( #IO.RunFwd )
      I_Contact( #IO.RunRev )
      I_Contact( #Pasue )
      Contact( #IO.HandStartSignal )
      Contact( #IO.InHand )
      { S7_Templates := "time_type := Time" } #GeneralDelayTimer.TON(pt := T#100MS, et =>)
      R_Coil( #IO.HandStartSignal )
   END_RUNG
   RUNG wire#powerrail
      I_Contact( #PreStartMemory )
   END_RUNG wire#w1
   // the same network as SCL:
   #IO.RecentStart := #IO.RecentStart AND NOT #IO.RunFwd AND NOT #IO.RunRev AND NOT #IO.FaultActive;
   #GeneralDelayTimer(IN := (NOT #IO.RecentStart OR NOT #PreStartMemory) AND NOT #IO.RunFwd AND NOT #IO.RunRev AND NOT #Pasue AND #IO.HandStartSignal AND #IO.InHand,   // TON
                      PT := T#100MS);
   IF #GeneralDelayTimer.Q THEN #IO.HandStartSignal := FALSE; END_IF;
END_REGION

REGION Network 5
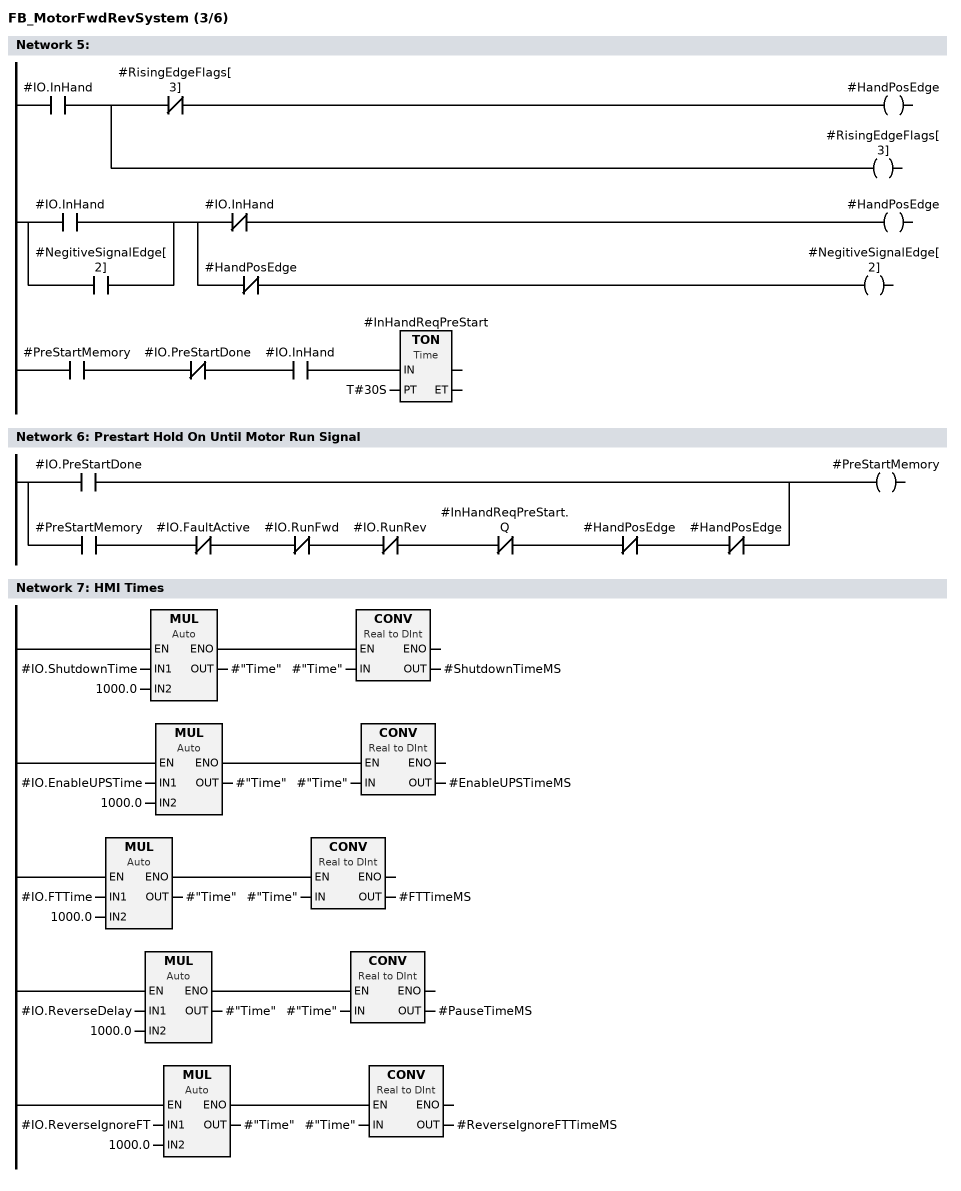
   RUNG wire#powerrail
      Contact( #IO.InHand )
      wire#w1
      I_Contact( #RisingEdgeFlags[3] )
      Coil( #HandPosEdge )
   END_RUNG
   RUNG wire#w1
      Coil( #RisingEdgeFlags[3] )
   END_RUNG
   RUNG wire#powerrail
      Contact( #IO.InHand )
      wire#w2
      I_Contact( #IO.InHand )
      Coil( #HandPosEdge )
   END_RUNG
   RUNG wire#powerrail
      Contact( #NegitiveSignalEdge[2] )
   END_RUNG wire#w2
   RUNG wire#w2
      I_Contact( #HandPosEdge )
      Coil( #NegitiveSignalEdge[2] )
   END_RUNG
   RUNG wire#powerrail
      Contact( #PreStartMemory )
      I_Contact( #IO.PreStartDone )
      Contact( #IO.InHand )
      { S7_Templates := "time_type := Time" } #InHandReqPreStart.TON(pt := T#30S, et =>)
   END_RUNG
   // the same network as SCL:
   #HandPosEdge := #IO.InHand AND NOT #RisingEdgeFlags[3];
   #RisingEdgeFlags[3] := #IO.InHand;
   #_w1 := #IO.InHand OR #NegitiveSignalEdge[2];
   #HandPosEdge := #_w1 AND NOT #IO.InHand;
   #NegitiveSignalEdge[2] := #_w1 AND NOT #HandPosEdge;
   #InHandReqPreStart(IN := #PreStartMemory AND NOT #IO.PreStartDone AND #IO.InHand, PT := T#30S);   // TON
END_REGION

REGION Network 6: Prestart Hold On Until Motor Run Signal
   RUNG wire#powerrail
      Contact( #IO.PreStartDone )
      wire#w1
      Coil( #PreStartMemory )
   END_RUNG
   RUNG wire#powerrail
      Contact( #PreStartMemory )
      I_Contact( #IO.FaultActive )
      I_Contact( #IO.RunFwd )
      I_Contact( #IO.RunRev )
      I_Contact( #InHandReqPreStart.Q )
      I_Contact( #HandPosEdge )
      I_Contact( #HandPosEdge )
   END_RUNG wire#w1
   // the same network as SCL:
   #PreStartMemory := #IO.PreStartDone OR (#PreStartMemory AND NOT #IO.FaultActive AND NOT #IO.RunFwd AND NOT #IO.RunRev AND NOT #InHandReqPreStart.Q AND NOT #HandPosEdge AND NOT #HandPosEdge);
END_REGION

REGION Network 7: HMI Times
   RUNG wire#powerrail
      Mul(in1 := #IO.ShutdownTime, in2 := 1000.0, out => #"Time")
      { S7_Templates := "[SrcType := Real, DestType := DInt]" } Convert(in := #"Time", out => #ShutdownTimeMS)
   END_RUNG
   RUNG wire#powerrail
      Mul(in1 := #IO.EnableUPSTime, in2 := 1000.0, out => #"Time")
      { S7_Templates := "[SrcType := Real, DestType := DInt]" } Convert(in := #"Time", out => #EnableUPSTimeMS)
   END_RUNG
   RUNG wire#powerrail
      Mul(in1 := #IO.FTTime, in2 := 1000.0, out => #"Time")
      { S7_Templates := "[SrcType := Real, DestType := DInt]" } Convert(in := #"Time", out => #FTTimeMS)
   END_RUNG
   RUNG wire#powerrail
      Mul(in1 := #IO.ReverseDelay, in2 := 1000.0, out => #"Time")
      { S7_Templates := "[SrcType := Real, DestType := DInt]" } Convert(in := #"Time", out => #PauseTimeMS)
   END_RUNG
   RUNG wire#powerrail
      Mul(in1 := #IO.ReverseIgnoreFT, in2 := 1000.0, out => #"Time")
      { S7_Templates := "[SrcType := Real, DestType := DInt]" } Convert(in := #"Time", out => #ReverseIgnoreFTTimeMS)
   END_RUNG
   // the same network as SCL:
   #"Time" := #IO.ShutdownTime * 1000.0;
   #ShutdownTimeMS := REAL_TO_DINT(#"Time");
   #"Time" := #IO.EnableUPSTime * 1000.0;
   #EnableUPSTimeMS := REAL_TO_DINT(#"Time");
   #"Time" := #IO.FTTime * 1000.0;
   #FTTimeMS := REAL_TO_DINT(#"Time");
   #"Time" := #IO.ReverseDelay * 1000.0;
   #PauseTimeMS := REAL_TO_DINT(#"Time");
   #"Time" := #IO.ReverseIgnoreFT * 1000.0;
   #ReverseIgnoreFTTimeMS := REAL_TO_DINT(#"Time");
END_REGION

REGION Network 8: DOL Motor Shutdown
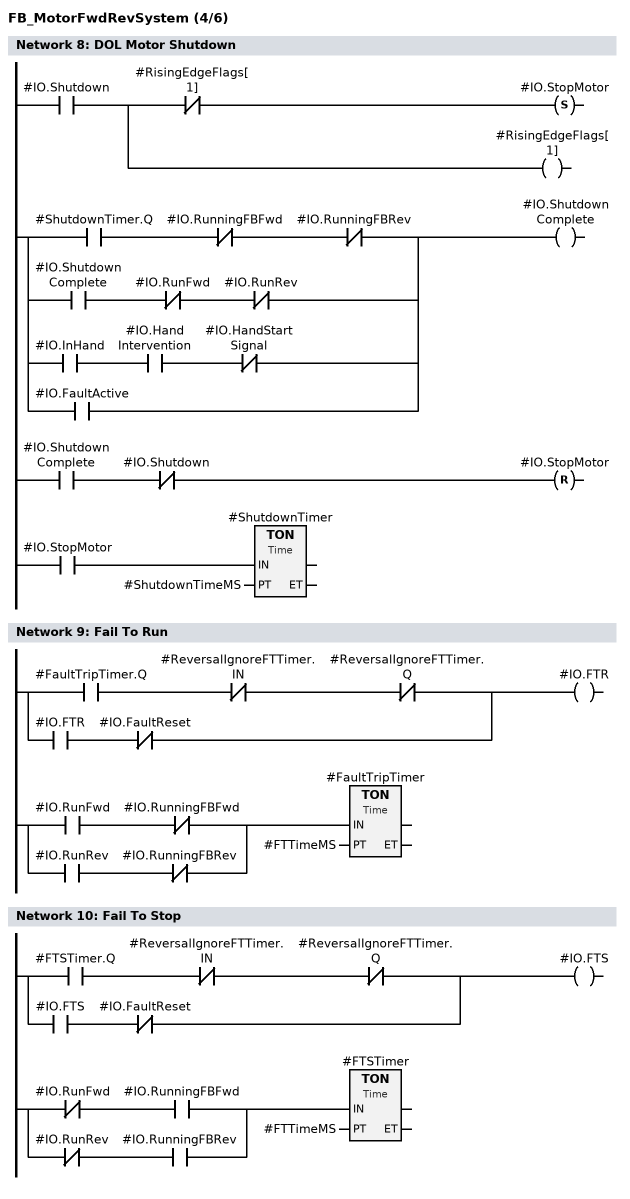
   RUNG wire#powerrail
      Contact( #IO.Shutdown )
      wire#w1
      I_Contact( #RisingEdgeFlags[1] )
      S_Coil( #IO.StopMotor )
   END_RUNG
   RUNG wire#w1
      Coil( #RisingEdgeFlags[1] )
   END_RUNG
   RUNG wire#powerrail
      Contact( #ShutdownTimer.Q )
      I_Contact( #IO.RunningFBFwd )
      I_Contact( #IO.RunningFBRev )
      wire#w2
      Coil( #IO.ShutdownComplete )
   END_RUNG
   RUNG wire#powerrail
      Contact( #IO.ShutdownComplete )
      I_Contact( #IO.RunFwd )
      I_Contact( #IO.RunRev )
   END_RUNG wire#w2
   RUNG wire#powerrail
      Contact( #IO.InHand )
      Contact( #IO.HandIntervention )
      I_Contact( #IO.HandStartSignal )
   END_RUNG wire#w2
   RUNG wire#powerrail
      Contact( #IO.FaultActive )
   END_RUNG wire#w2
   RUNG wire#powerrail
      Contact( #IO.ShutdownComplete )
      I_Contact( #IO.Shutdown )
      R_Coil( #IO.StopMotor )
   END_RUNG
   RUNG wire#powerrail
      Contact( #IO.StopMotor )
      { S7_Templates := "time_type := Time" } #ShutdownTimer.TON(pt := #ShutdownTimeMS, et =>)
   END_RUNG
   // the same network as SCL:
   IF #IO.Shutdown AND NOT #RisingEdgeFlags[1] THEN #IO.StopMotor := TRUE; END_IF;
   #RisingEdgeFlags[1] := #IO.Shutdown;
   #IO.ShutdownComplete := (#ShutdownTimer.Q AND NOT #IO.RunningFBFwd AND NOT #IO.RunningFBRev) OR (#IO.ShutdownComplete AND NOT #IO.RunFwd AND NOT #IO.RunRev) OR (#IO.InHand AND #IO.HandIntervention AND NOT #IO.HandStartSignal) OR #IO.FaultActive;
   IF #IO.ShutdownComplete AND NOT #IO.Shutdown THEN #IO.StopMotor := FALSE; END_IF;
   #ShutdownTimer(IN := #IO.StopMotor, PT := #ShutdownTimeMS);   // TON
END_REGION

REGION Network 9: Fail To Run
   RUNG wire#powerrail
      Contact( #FaultTripTimer.Q )
      I_Contact( #ReversalIgnoreFTTimer.IN )
      I_Contact( #ReversalIgnoreFTTimer.Q )
      wire#w1
      Coil( #IO.FTR )
   END_RUNG
   RUNG wire#powerrail
      Contact( #IO.FTR )
      I_Contact( #IO.FaultReset )
   END_RUNG wire#w1
   RUNG wire#powerrail
      Contact( #IO.RunFwd )
      I_Contact( #IO.RunningFBFwd )
      wire#w2
      { S7_Templates := "time_type := Time" } #FaultTripTimer.TON(pt := #FTTimeMS, et =>)
   END_RUNG
   RUNG wire#powerrail
      Contact( #IO.RunRev )
      I_Contact( #IO.RunningFBRev )
   END_RUNG wire#w2
   // the same network as SCL:
   #IO.FTR := (#FaultTripTimer.Q AND NOT #ReversalIgnoreFTTimer.IN AND NOT #ReversalIgnoreFTTimer.Q) OR (#IO.FTR AND NOT #IO.FaultReset);
   #FaultTripTimer(IN := (#IO.RunFwd AND NOT #IO.RunningFBFwd) OR (#IO.RunRev AND NOT #IO.RunningFBRev),   // TON
                   PT := #FTTimeMS);
END_REGION

REGION Network 10: Fail To Stop
   RUNG wire#powerrail
      Contact( #FTSTimer.Q )
      I_Contact( #ReversalIgnoreFTTimer.IN )
      I_Contact( #ReversalIgnoreFTTimer.Q )
      wire#w1
      Coil( #IO.FTS )
   END_RUNG
   RUNG wire#powerrail
      Contact( #IO.FTS )
      I_Contact( #IO.FaultReset )
   END_RUNG wire#w1
   RUNG wire#powerrail
      I_Contact( #IO.RunFwd )
      Contact( #IO.RunningFBFwd )
      wire#w2
      { S7_Templates := "time_type := Time" } #FTSTimer.TON(pt := #FTTimeMS, et =>)
   END_RUNG
   RUNG wire#powerrail
      I_Contact( #IO.RunRev )
      Contact( #IO.RunningFBRev )
   END_RUNG wire#w2
   // the same network as SCL:
   #IO.FTS := (#FTSTimer.Q AND NOT #ReversalIgnoreFTTimer.IN AND NOT #ReversalIgnoreFTTimer.Q) OR (#IO.FTS AND NOT #IO.FaultReset);
   #FTSTimer(IN := (NOT #IO.RunFwd AND #IO.RunningFBFwd) OR (NOT #IO.RunRev AND #IO.RunningFBRev),   // TON
             PT := #FTTimeMS);
END_REGION

REGION Network 11: Faults
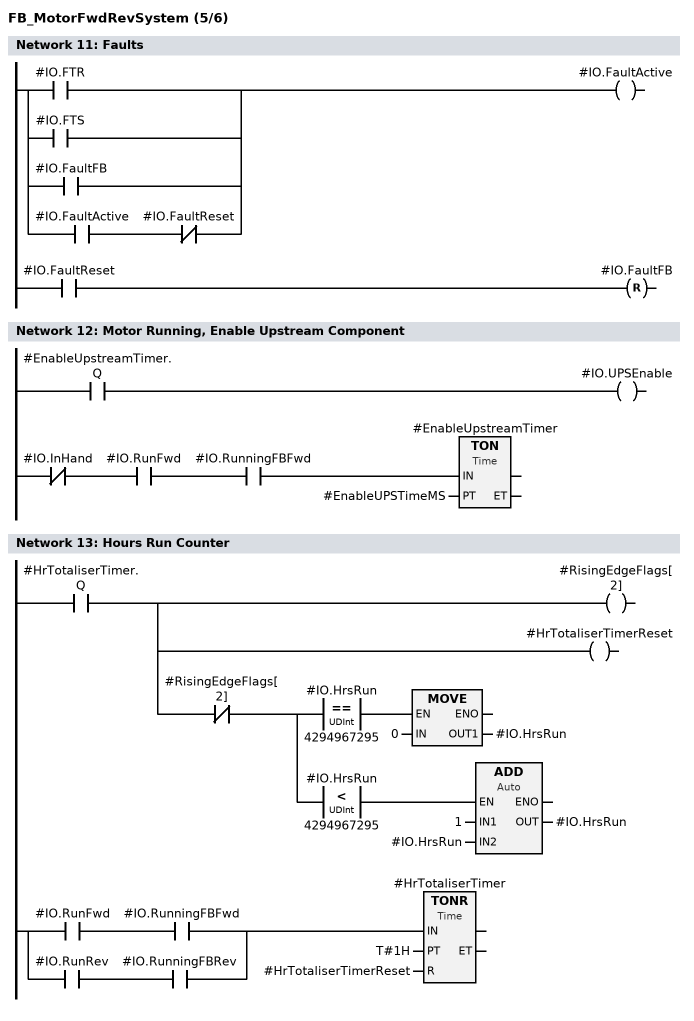
   RUNG wire#powerrail
      Contact( #IO.FTR )
      wire#w1
      Coil( #IO.FaultActive )
   END_RUNG
   RUNG wire#powerrail
      Contact( #IO.FTS )
   END_RUNG wire#w1
   RUNG wire#powerrail
      Contact( #IO.FaultFB )
   END_RUNG wire#w1
   RUNG wire#powerrail
      Contact( #IO.FaultActive )
      I_Contact( #IO.FaultReset )
   END_RUNG wire#w1
   RUNG wire#powerrail
      Contact( #IO.FaultReset )
      R_Coil( #IO.FaultFB )
   END_RUNG
   // the same network as SCL:
   #IO.FaultActive := #IO.FTR OR #IO.FTS OR #IO.FaultFB OR (#IO.FaultActive AND NOT #IO.FaultReset);
   IF #IO.FaultReset THEN #IO.FaultFB := FALSE; END_IF;
END_REGION

REGION Network 12: Motor Running, Enable Upstream Component
   RUNG wire#powerrail
      Contact( #EnableUpstreamTimer.Q )
      Coil( #IO.UPSEnable )
   END_RUNG
   RUNG wire#powerrail
      I_Contact( #IO.InHand )
      Contact( #IO.RunFwd )
      Contact( #IO.RunningFBFwd )
      { S7_Templates := "time_type := Time" } #EnableUpstreamTimer.TON(pt := #EnableUPSTimeMS, et =>)
   END_RUNG
   // the same network as SCL:
   #IO.UPSEnable := #EnableUpstreamTimer.Q;
   #EnableUpstreamTimer(IN := NOT #IO.InHand AND #IO.RunFwd AND #IO.RunningFBFwd, PT := #EnableUPSTimeMS);   // TON
END_REGION

REGION Network 13: Hours Run Counter
   RUNG wire#powerrail
      Contact( #HrTotaliserTimer.Q )
      wire#w1
      Coil( #RisingEdgeFlags[2] )
   END_RUNG
   RUNG wire#w1
      Coil( #HrTotaliserTimerReset )
   END_RUNG
   RUNG wire#w1
      I_Contact( #RisingEdgeFlags[2] )
      wire#w2
      { S7_Templates := "SrcType := UDInt" } EQ_Contact(in1 := #IO.HrsRun, in2 := 4294967295)
      Move(in := 0, out1 => #IO.HrsRun)
   END_RUNG
   RUNG wire#w2
      { S7_Templates := "SrcType := UDInt" } LT_Contact(in1 := #IO.HrsRun, in2 := 4294967295)
      Add(in1 := 1, in2 := #IO.HrsRun, out => #IO.HrsRun)
   END_RUNG
   RUNG wire#powerrail
      Contact( #IO.RunFwd )
      Contact( #IO.RunningFBFwd )
      wire#w3
      { S7_Templates := "time_type := Time" } #HrTotaliserTimer.TONR(pt := T#1H, et =>, r := #HrTotaliserTimerReset)
   END_RUNG
   RUNG wire#powerrail
      Contact( #IO.RunRev )
      Contact( #IO.RunningFBRev )
   END_RUNG wire#w3
   // the same network as SCL:
   #RisingEdgeFlags[2] := #HrTotaliserTimer.Q;
   #HrTotaliserTimerReset := #HrTotaliserTimer.Q;
   #_w1 := #HrTotaliserTimer.Q AND NOT #RisingEdgeFlags[2];
   IF #_w1 AND (#IO.HrsRun = 4294967295) THEN #IO.HrsRun := 0; END_IF;
   IF #_w1 AND (#IO.HrsRun < 4294967295) THEN #IO.HrsRun := 1 + #IO.HrsRun; END_IF;
   #HrTotaliserTimer(IN := (#IO.RunFwd AND #IO.RunningFBFwd) OR (#IO.RunRev AND #IO.RunningFBRev),   // TONR
                     PT := T#1H,
                     R := #HrTotaliserTimerReset);
END_REGION

REGION Network 14: HMI Motor Status Telemetry
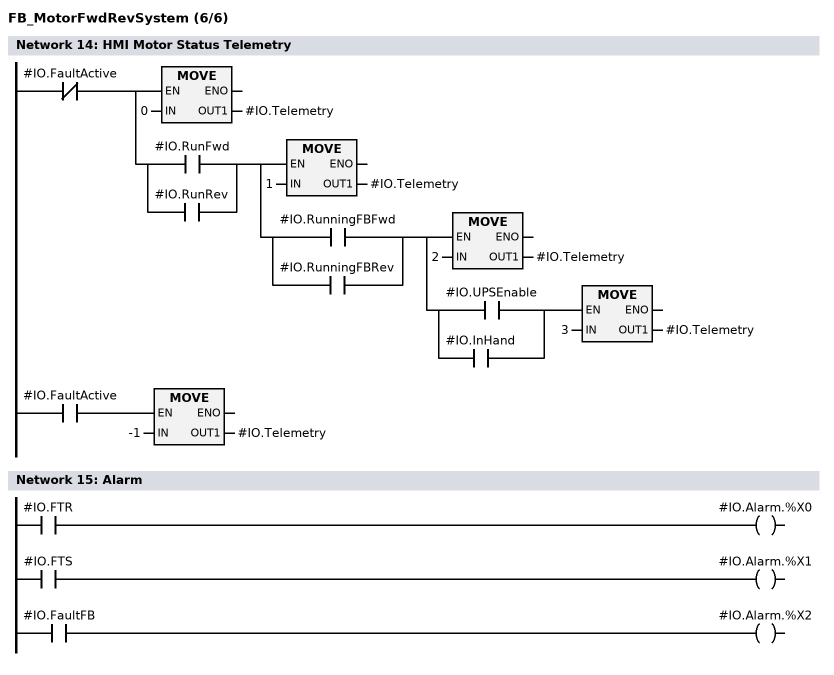
   RUNG wire#powerrail
      I_Contact( #IO.FaultActive )
      wire#w1
      Move(in := 0, out1 => #IO.Telemetry)
   END_RUNG
   RUNG wire#w1
      Contact( #IO.RunFwd )
      wire#w2
      Move(in := 1, out1 => #IO.Telemetry)
   END_RUNG
   RUNG wire#w1
      Contact( #IO.RunRev )
   END_RUNG wire#w2
   RUNG wire#w2
      Contact( #IO.RunningFBFwd )
      wire#w3
      Move(in := 2, out1 => #IO.Telemetry)
   END_RUNG
   RUNG wire#w2
      Contact( #IO.RunningFBRev )
   END_RUNG wire#w3
   RUNG wire#w3
      Contact( #IO.UPSEnable )
      wire#w4
      Move(in := 3, out1 => #IO.Telemetry)
   END_RUNG
   RUNG wire#w3
      Contact( #IO.InHand )
   END_RUNG wire#w4
   RUNG wire#powerrail
      Contact( #IO.FaultActive )
      Move(in := -1, out1 => #IO.Telemetry)
   END_RUNG
   // the same network as SCL:
   IF NOT #IO.FaultActive THEN #IO.Telemetry := 0; END_IF;
   #_w1 := NOT #IO.FaultActive AND (#IO.RunFwd OR #IO.RunRev);
   IF #_w1 THEN #IO.Telemetry := 1; END_IF;
   #_w2 := #_w1 AND (#IO.RunningFBFwd OR #IO.RunningFBRev);
   IF #_w2 THEN #IO.Telemetry := 2; END_IF;
   IF #_w2 AND (#IO.UPSEnable OR #IO.InHand) THEN #IO.Telemetry := 3; END_IF;
   IF #IO.FaultActive THEN #IO.Telemetry := -1; END_IF;
END_REGION

REGION Network 15: Alarm
   RUNG wire#powerrail
      Contact( #IO.FTR )
      Coil( #IO.Alarm.%X0 )
   END_RUNG
   RUNG wire#powerrail
      Contact( #IO.FTS )
      Coil( #IO.Alarm.%X1 )
   END_RUNG
   RUNG wire#powerrail
      Contact( #IO.FaultFB )
      Coil( #IO.Alarm.%X2 )
   END_RUNG
   // the same network as SCL:
   #IO.Alarm.%X0 := #IO.FTR;
   #IO.Alarm.%X1 := #IO.FTS;
   #IO.Alarm.%X2 := #IO.FaultFB;
END_REGION
END_FUNCTION_BLOCK

FUNCTION_BLOCK "FB_PusherControl"   // FB3, LAD
TITLE = Pusher Control
{ S7_Optimized_Access := 'TRUE' }
VERSION : 0.1
// Pusher ram sequencing (C-118-C-125). Step legend (C-120): 0=Parked (idle/home, ram fully retracted, no motion) - 10=DriveToEndTravel (forward stroke in progress) - 20=Hold (paused at full travel, brief settle before retracting) - 30=Retract (returning to home; also the recovery/abort target from any bad state). Mode legend: 0=Off (finish a retract already in progress, then park; no new cycle starts) - 1=Auto (hopper-high-level starts a cycle) - 2=Manual (operator button/jog starts a cycle).
// stored: AutoNumber true, IsIECCheckEnabled false, IsRetainMemResEnabled false, MemoryReserve 100, SetENOAutomatically false, UDAEnableTagReadback false
   VAR RETAIN
      IO { S7_SetPoint := 'True'} : "UDT_PusherIO";   // Caller-visible interface (C-115) - FC_ControlMain writes Mode/HopperHighLevel/limits/tunables in, reads Extend/Retract/RunPowerPack/fault bits out. See the block header for the Step/Mode value legend.
   END_VAR
   VAR
      EndTravelTimeoutMS : DInt;
      ParkedTimeoutMS : DInt;
      EndTravelHoldTimeMS : DInt;
      PumpRunOnTimeMS : DInt;
      JogWarningTimeMS : DInt;
      PressureTripConfirmTimeMS : DInt;
      PressureClearResumeDelayMS : DInt;
      PressureConfirmTimer { S7_SetPoint := 'True'} : TON_TIME;
      PressureClearTimer { S7_SetPoint := 'True'} : TON_TIME;
      PressureHold : Bool;   // Latched jam hold, not a fault (C-123) - see the Pressure Detection network. Freezes ExtendDemand while set; clears itself once pressure has genuinely stayed clear for PressureClearResumeDelay.
      PressureConfirmEdge : Bool;
      PressureConfirmEdgeMem : Bool;
      PressureTripCount : Int;   // Confirmed jams this cycle - reset each cycle start, not time-windowed. Compared against IO.PressureTripCountThreshold to raise Blocked.
      EndTravelTimer { S7_SetPoint := 'True'} : TON_TIME;
      HoldTimer { S7_SetPoint := 'True'} : TON_TIME;
      ParkedTimer { S7_SetPoint := 'True'} : TON_TIME;
      JogPreStartTimer { S7_SetPoint := 'True'} : TON_TIME;
      ExtendDemand : Bool;
      RetractDemand : Bool;
      PumpDemand : Bool;   // ExtendDemand OR RetractDemand - the pump's own immediate (non-run-on) demand signal.
      PumpEverDemanded : Bool;   // Cold-start guard for the pump run-on off-delay below - see that network's own comment.
      PumpRunOnTimer { S7_SetPoint := 'True'} : TON_TIME;
   END_VAR
   VAR_TEMP
      "Time" : Real;
   END_VAR
BEGIN

REGION Network 1: Enable
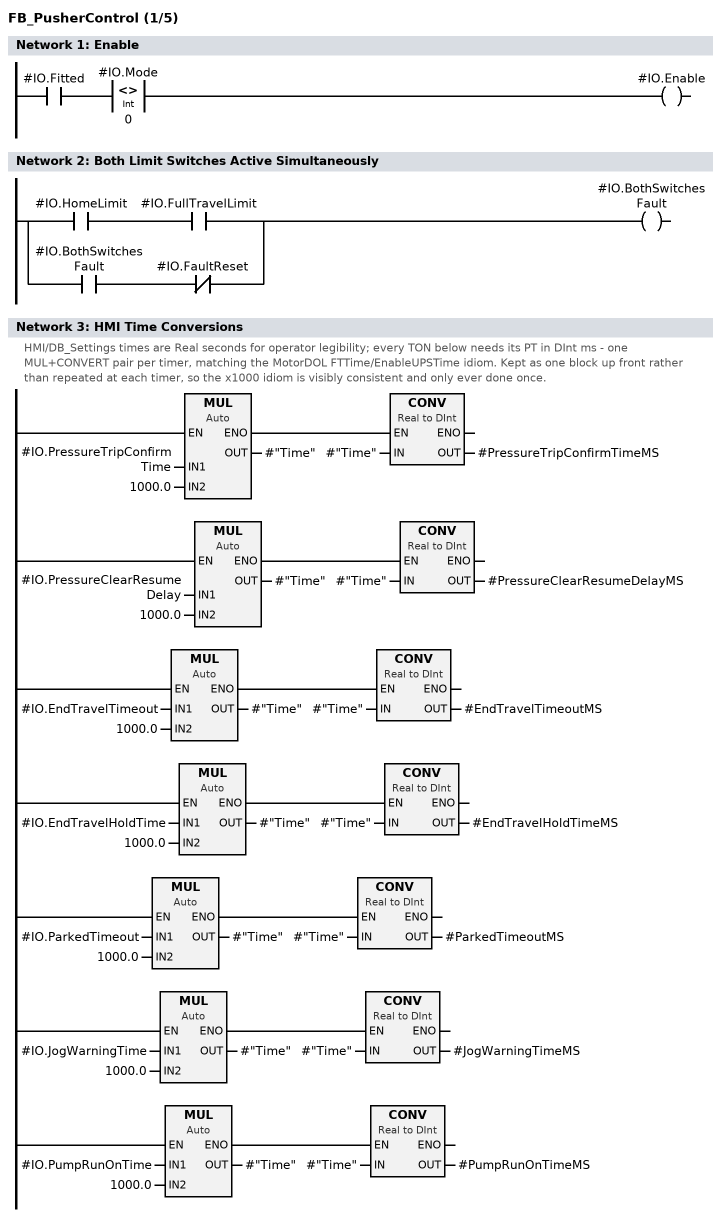
   RUNG wire#powerrail
      Contact( #IO.Fitted )
      { S7_Templates := "SrcType := Int" } NE_Contact(in1 := #IO.Mode, in2 := 0)
      Coil( #IO.Enable )
   END_RUNG
   // the same network as SCL:
   #IO.Enable := #IO.Fitted AND (#IO.Mode <> 0);
END_REGION

REGION Network 2: Both Limit Switches Active Simultaneously
   RUNG wire#powerrail
      Contact( #IO.HomeLimit )
      Contact( #IO.FullTravelLimit )
      wire#w1
      Coil( #IO.BothSwitchesFault )
   END_RUNG
   RUNG wire#powerrail
      Contact( #IO.BothSwitchesFault )
      I_Contact( #IO.FaultReset )
   END_RUNG wire#w1
   // the same network as SCL:
   #IO.BothSwitchesFault := (#IO.HomeLimit AND #IO.FullTravelLimit) OR (#IO.BothSwitchesFault AND NOT #IO.FaultReset);
END_REGION

REGION Network 3: HMI Time Conversions
   // HMI/DB_Settings times are Real seconds for operator legibility; every TON below needs its PT in DInt ms - one MUL+CONVERT pair per timer, matching the MotorDOL FTTime/EnableUPSTime idiom. Kept as one block up front rather than repeated at each timer, so the x1000 idiom is visibly consistent and only ever done once.
   RUNG wire#powerrail
      Mul(in1 := #IO.PressureTripConfirmTime, in2 := 1000.0, out => #"Time")
      { S7_Templates := "[SrcType := Real, DestType := DInt]" } Convert(in := #"Time", out => #PressureTripConfirmTimeMS)
   END_RUNG
   RUNG wire#powerrail
      Mul(in1 := #IO.PressureClearResumeDelay, in2 := 1000.0, out => #"Time")
      { S7_Templates := "[SrcType := Real, DestType := DInt]" } Convert(in := #"Time", out => #PressureClearResumeDelayMS)
   END_RUNG
   RUNG wire#powerrail
      Mul(in1 := #IO.EndTravelTimeout, in2 := 1000.0, out => #"Time")
      { S7_Templates := "[SrcType := Real, DestType := DInt]" } Convert(in := #"Time", out => #EndTravelTimeoutMS)
   END_RUNG
   RUNG wire#powerrail
      Mul(in1 := #IO.EndTravelHoldTime, in2 := 1000.0, out => #"Time")
      { S7_Templates := "[SrcType := Real, DestType := DInt]" } Convert(in := #"Time", out => #EndTravelHoldTimeMS)
   END_RUNG
   RUNG wire#powerrail
      Mul(in1 := #IO.ParkedTimeout, in2 := 1000.0, out => #"Time")
      { S7_Templates := "[SrcType := Real, DestType := DInt]" } Convert(in := #"Time", out => #ParkedTimeoutMS)
   END_RUNG
   RUNG wire#powerrail
      Mul(in1 := #IO.JogWarningTime, in2 := 1000.0, out => #"Time")
      { S7_Templates := "[SrcType := Real, DestType := DInt]" } Convert(in := #"Time", out => #JogWarningTimeMS)
   END_RUNG
   RUNG wire#powerrail
      Mul(in1 := #IO.PumpRunOnTime, in2 := 1000.0, out => #"Time")
      { S7_Templates := "[SrcType := Real, DestType := DInt]" } Convert(in := #"Time", out => #PumpRunOnTimeMS)
   END_RUNG
   // the same network as SCL:
   #"Time" := #IO.PressureTripConfirmTime * 1000.0;
   #PressureTripConfirmTimeMS := REAL_TO_DINT(#"Time");
   #"Time" := #IO.PressureClearResumeDelay * 1000.0;
   #PressureClearResumeDelayMS := REAL_TO_DINT(#"Time");
   #"Time" := #IO.EndTravelTimeout * 1000.0;
   #EndTravelTimeoutMS := REAL_TO_DINT(#"Time");
   #"Time" := #IO.EndTravelHoldTime * 1000.0;
   #EndTravelHoldTimeMS := REAL_TO_DINT(#"Time");
   #"Time" := #IO.ParkedTimeout * 1000.0;
   #ParkedTimeoutMS := REAL_TO_DINT(#"Time");
   #"Time" := #IO.JogWarningTime * 1000.0;
   #JogWarningTimeMS := REAL_TO_DINT(#"Time");
   #"Time" := #IO.PumpRunOnTime * 1000.0;
   #PumpRunOnTimeMS := REAL_TO_DINT(#"Time");
END_REGION

REGION Network 4: Pressure Trip Detection, Hold, And Counting
   // One function, one network: a trip must be debounced (PressureConfirmTimer) before it counts - momentary pressure spikes aren't a real jam. Hold latches through a confirmed trip and only releases once pressure has genuinely cleared for PressureClearResumeDelay, so a bouncing switch can't re-trigger the count on every scan. Count resets each cycle start (Step 0-to-10 launch condition), not on a rolling time window.
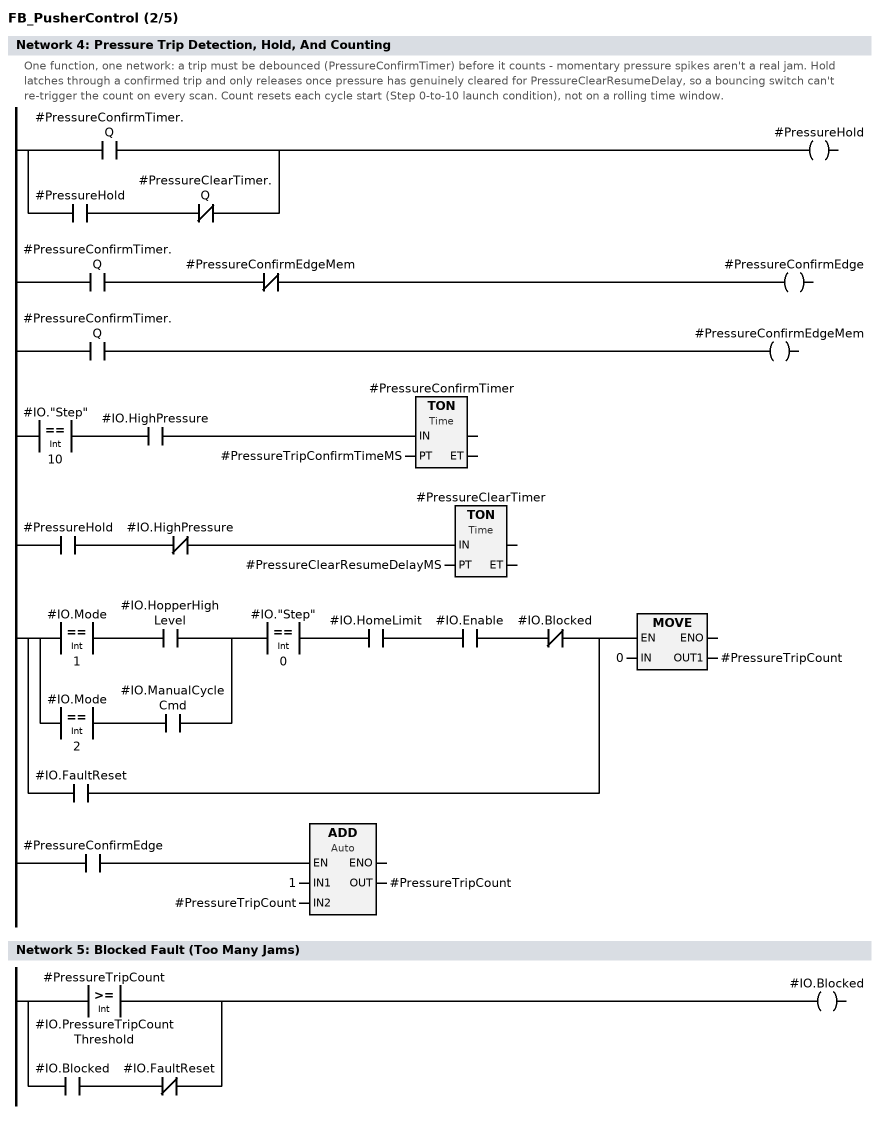
   RUNG wire#powerrail
      Contact( #PressureConfirmTimer.Q )
      wire#w1
      Coil( #PressureHold )
   END_RUNG
   RUNG wire#powerrail
      Contact( #PressureHold )
      I_Contact( #PressureClearTimer.Q )
   END_RUNG wire#w1
   RUNG wire#powerrail
      Contact( #PressureConfirmTimer.Q )
      I_Contact( #PressureConfirmEdgeMem )
      Coil( #PressureConfirmEdge )
   END_RUNG
   RUNG wire#powerrail
      Contact( #PressureConfirmTimer.Q )
      Coil( #PressureConfirmEdgeMem )
   END_RUNG
   RUNG wire#powerrail
      { S7_Templates := "SrcType := Int" } EQ_Contact(in1 := #IO."Step", in2 := 10)
      Contact( #IO.HighPressure )
      { S7_Templates := "time_type := Time" } #PressureConfirmTimer.TON(pt := #PressureTripConfirmTimeMS, et =>)
   END_RUNG
   RUNG wire#powerrail
      Contact( #PressureHold )
      I_Contact( #IO.HighPressure )
      { S7_Templates := "time_type := Time" } #PressureClearTimer.TON(pt := #PressureClearResumeDelayMS, et =>)
   END_RUNG
   RUNG wire#powerrail
      { S7_Templates := "SrcType := Int" } EQ_Contact(in1 := #IO.Mode, in2 := 1)
      Contact( #IO.HopperHighLevel )
      wire#w2
      { S7_Templates := "SrcType := Int" } EQ_Contact(in1 := #IO."Step", in2 := 0)
      Contact( #IO.HomeLimit )
      Contact( #IO.Enable )
      I_Contact( #IO.Blocked )
      wire#w3
      Move(in := 0, out1 => #PressureTripCount)
   END_RUNG
   RUNG wire#powerrail
      { S7_Templates := "SrcType := Int" } EQ_Contact(in1 := #IO.Mode, in2 := 2)
      Contact( #IO.ManualCycleCmd )
   END_RUNG wire#w2
   RUNG wire#powerrail
      Contact( #IO.FaultReset )
   END_RUNG wire#w3
   RUNG wire#powerrail
      Contact( #PressureConfirmEdge )
      Add(in1 := 1, in2 := #PressureTripCount, out => #PressureTripCount)
   END_RUNG
   // the same network as SCL:
   #PressureHold := #PressureConfirmTimer.Q OR (#PressureHold AND NOT #PressureClearTimer.Q);
   #PressureConfirmEdge := #PressureConfirmTimer.Q AND NOT #PressureConfirmEdgeMem;
   #PressureConfirmEdgeMem := #PressureConfirmTimer.Q;
   #PressureConfirmTimer(IN := (#IO."Step" = 10) AND #IO.HighPressure, PT := #PressureTripConfirmTimeMS);   // TON
   #PressureClearTimer(IN := #PressureHold AND NOT #IO.HighPressure, PT := #PressureClearResumeDelayMS);   // TON
   IF ((((#IO.Mode = 1) AND #IO.HopperHighLevel) OR ((#IO.Mode = 2) AND #IO.ManualCycleCmd)) AND (#IO."Step" = 0) AND #IO.HomeLimit AND #IO.Enable AND NOT #IO.Blocked) OR #IO.FaultReset THEN
       #PressureTripCount := 0;
   END_IF;
   IF #PressureConfirmEdge THEN #PressureTripCount := 1 + #PressureTripCount; END_IF;
END_REGION

REGION Network 5: Blocked Fault (Too Many Jams)
   RUNG wire#powerrail
      { S7_Templates := "SrcType := Int" } GE_Contact(in1 := #PressureTripCount, in2 := #IO.PressureTripCountThreshold)
      wire#w1
      Coil( #IO.Blocked )
   END_RUNG
   RUNG wire#powerrail
      Contact( #IO.Blocked )
      I_Contact( #IO.FaultReset )
   END_RUNG wire#w1
   // the same network as SCL:
   #IO.Blocked := (#PressureTripCount >= #IO.PressureTripCountThreshold) OR (#IO.Blocked AND NOT #IO.FaultReset);
END_REGION

REGION Network 6: Step 0 (Parked) - Transitions
   // Not-at-home while idle (power-up mid-stroke, or a cycle that ended without reaching HomeLimit) drives straight to Retract (30) to re-establish home before any new cycle is accepted - never straight back into a forward stroke from an unknown position. Suppressed during an active jog command so jogging isn't fought by an auto-retract.
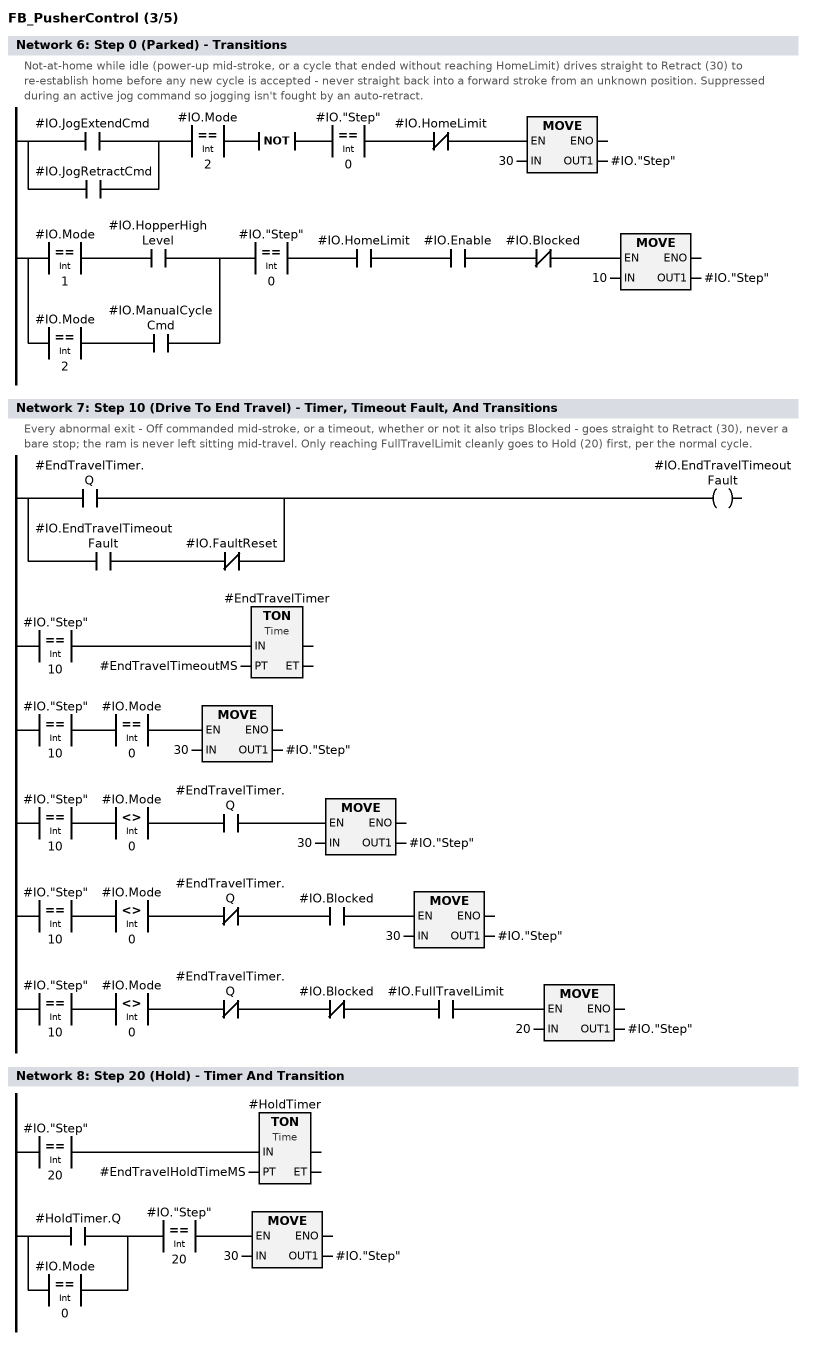
   RUNG wire#powerrail
      Contact( #IO.JogExtendCmd )
      wire#w1
      { S7_Templates := "SrcType := Int" } EQ_Contact(in1 := #IO.Mode, in2 := 2)
      Not()
      { S7_Templates := "SrcType := Int" } EQ_Contact(in1 := #IO."Step", in2 := 0)
      I_Contact( #IO.HomeLimit )
      Move(in := 30, out1 => #IO."Step")
   END_RUNG
   RUNG wire#powerrail
      Contact( #IO.JogRetractCmd )
   END_RUNG wire#w1
   RUNG wire#powerrail
      { S7_Templates := "SrcType := Int" } EQ_Contact(in1 := #IO.Mode, in2 := 1)
      Contact( #IO.HopperHighLevel )
      wire#w2
      { S7_Templates := "SrcType := Int" } EQ_Contact(in1 := #IO."Step", in2 := 0)
      Contact( #IO.HomeLimit )
      Contact( #IO.Enable )
      I_Contact( #IO.Blocked )
      Move(in := 10, out1 => #IO."Step")
   END_RUNG
   RUNG wire#powerrail
      { S7_Templates := "SrcType := Int" } EQ_Contact(in1 := #IO.Mode, in2 := 2)
      Contact( #IO.ManualCycleCmd )
   END_RUNG wire#w2
   // the same network as SCL:
   IF NOT ((#IO.JogExtendCmd OR #IO.JogRetractCmd) AND (#IO.Mode = 2)) AND (#IO."Step" = 0) AND NOT #IO.HomeLimit THEN
       #IO."Step" := 30;
   END_IF;
   IF (((#IO.Mode = 1) AND #IO.HopperHighLevel) OR ((#IO.Mode = 2) AND #IO.ManualCycleCmd)) AND (#IO."Step" = 0) AND #IO.HomeLimit AND #IO.Enable AND NOT #IO.Blocked THEN
       #IO."Step" := 10;
   END_IF;
END_REGION

REGION Network 7: Step 10 (Drive To End Travel) - Timer, Timeout Fault, And Transitions
   // Every abnormal exit - Off commanded mid-stroke, or a timeout, whether or not it also trips Blocked - goes straight to Retract (30), never a bare stop; the ram is never left sitting mid-travel. Only reaching FullTravelLimit cleanly goes to Hold (20) first, per the normal cycle.
   RUNG wire#powerrail
      Contact( #EndTravelTimer.Q )
      wire#w1
      Coil( #IO.EndTravelTimeoutFault )
   END_RUNG
   RUNG wire#powerrail
      Contact( #IO.EndTravelTimeoutFault )
      I_Contact( #IO.FaultReset )
   END_RUNG wire#w1
   RUNG wire#powerrail
      { S7_Templates := "SrcType := Int" } EQ_Contact(in1 := #IO."Step", in2 := 10)
      { S7_Templates := "time_type := Time" } #EndTravelTimer.TON(pt := #EndTravelTimeoutMS, et =>)
   END_RUNG
   RUNG wire#powerrail
      { S7_Templates := "SrcType := Int" } EQ_Contact(in1 := #IO."Step", in2 := 10)
      { S7_Templates := "SrcType := Int" } EQ_Contact(in1 := #IO.Mode, in2 := 0)
      Move(in := 30, out1 => #IO."Step")
   END_RUNG
   RUNG wire#powerrail
      { S7_Templates := "SrcType := Int" } EQ_Contact(in1 := #IO."Step", in2 := 10)
      { S7_Templates := "SrcType := Int" } NE_Contact(in1 := #IO.Mode, in2 := 0)
      Contact( #EndTravelTimer.Q )
      Move(in := 30, out1 => #IO."Step")
   END_RUNG
   RUNG wire#powerrail
      { S7_Templates := "SrcType := Int" } EQ_Contact(in1 := #IO."Step", in2 := 10)
      { S7_Templates := "SrcType := Int" } NE_Contact(in1 := #IO.Mode, in2 := 0)
      I_Contact( #EndTravelTimer.Q )
      Contact( #IO.Blocked )
      Move(in := 30, out1 => #IO."Step")
   END_RUNG
   RUNG wire#powerrail
      { S7_Templates := "SrcType := Int" } EQ_Contact(in1 := #IO."Step", in2 := 10)
      { S7_Templates := "SrcType := Int" } NE_Contact(in1 := #IO.Mode, in2 := 0)
      I_Contact( #EndTravelTimer.Q )
      I_Contact( #IO.Blocked )
      Contact( #IO.FullTravelLimit )
      Move(in := 20, out1 => #IO."Step")
   END_RUNG
   // the same network as SCL:
   #IO.EndTravelTimeoutFault := #EndTravelTimer.Q OR (#IO.EndTravelTimeoutFault AND NOT #IO.FaultReset);
   #EndTravelTimer(IN := #IO."Step" = 10, PT := #EndTravelTimeoutMS);   // TON
   IF (#IO."Step" = 10) AND (#IO.Mode = 0) THEN #IO."Step" := 30; END_IF;
   IF (#IO."Step" = 10) AND (#IO.Mode <> 0) AND #EndTravelTimer.Q THEN #IO."Step" := 30; END_IF;
   IF (#IO."Step" = 10) AND (#IO.Mode <> 0) AND NOT #EndTravelTimer.Q AND #IO.Blocked THEN
       #IO."Step" := 30;
   END_IF;
   IF (#IO."Step" = 10) AND (#IO.Mode <> 0) AND NOT #EndTravelTimer.Q AND NOT #IO.Blocked AND #IO.FullTravelLimit THEN
       #IO."Step" := 20;
   END_IF;
END_REGION

REGION Network 8: Step 20 (Hold) - Timer And Transition
   RUNG wire#powerrail
      { S7_Templates := "SrcType := Int" } EQ_Contact(in1 := #IO."Step", in2 := 20)
      { S7_Templates := "time_type := Time" } #HoldTimer.TON(pt := #EndTravelHoldTimeMS, et =>)
   END_RUNG
   RUNG wire#powerrail
      Contact( #HoldTimer.Q )
      wire#w1
      { S7_Templates := "SrcType := Int" } EQ_Contact(in1 := #IO."Step", in2 := 20)
      Move(in := 30, out1 => #IO."Step")
   END_RUNG
   RUNG wire#powerrail
      { S7_Templates := "SrcType := Int" } EQ_Contact(in1 := #IO.Mode, in2 := 0)
   END_RUNG wire#w1
   // the same network as SCL:
   #HoldTimer(IN := #IO."Step" = 20, PT := #EndTravelHoldTimeMS);   // TON
   IF (#HoldTimer.Q OR (#IO.Mode = 0)) AND (#IO."Step" = 20) THEN #IO."Step" := 30; END_IF;
END_REGION

REGION Network 9: Step 30 (Retract) - Timer, Timeout Fault, And Transition
   // ParkedTimer's own Q only feeds the timeout fault, not a transition - if genuinely stuck retracting there's no safer step to force (unlike Step 10, nothing here can be aborted into); alarm-only by design, awaiting a human.
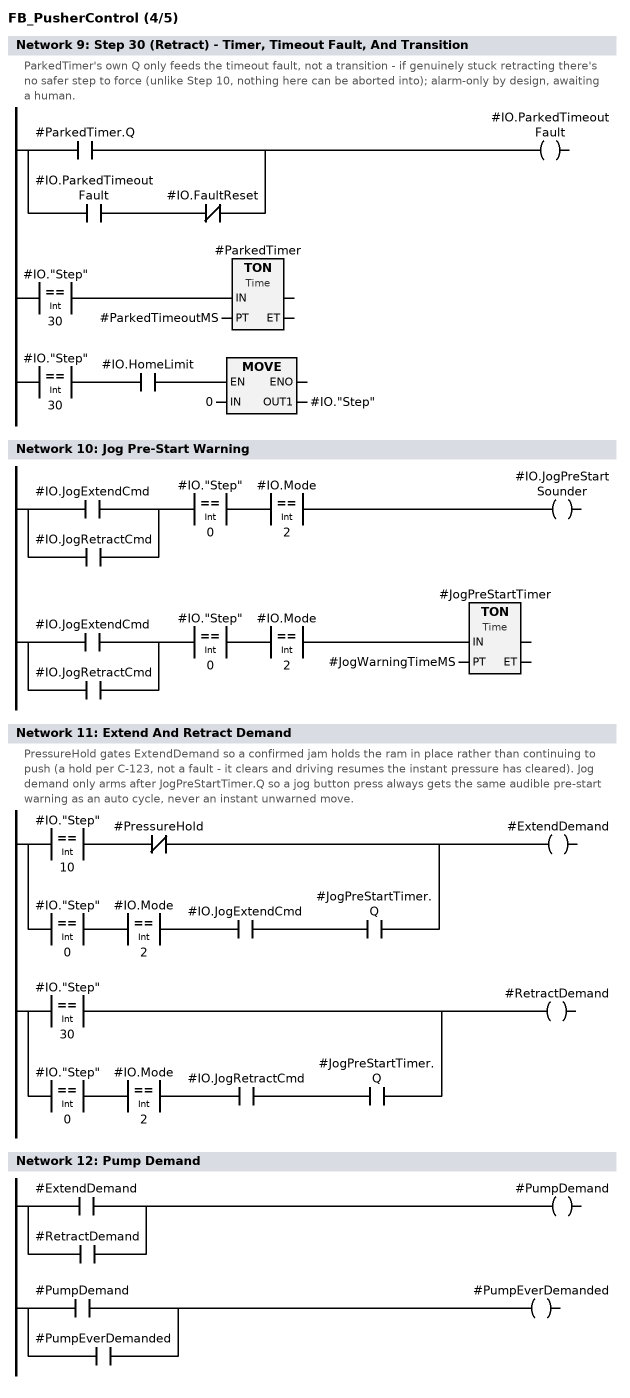
   RUNG wire#powerrail
      Contact( #ParkedTimer.Q )
      wire#w1
      Coil( #IO.ParkedTimeoutFault )
   END_RUNG
   RUNG wire#powerrail
      Contact( #IO.ParkedTimeoutFault )
      I_Contact( #IO.FaultReset )
   END_RUNG wire#w1
   RUNG wire#powerrail
      { S7_Templates := "SrcType := Int" } EQ_Contact(in1 := #IO."Step", in2 := 30)
      { S7_Templates := "time_type := Time" } #ParkedTimer.TON(pt := #ParkedTimeoutMS, et =>)
   END_RUNG
   RUNG wire#powerrail
      { S7_Templates := "SrcType := Int" } EQ_Contact(in1 := #IO."Step", in2 := 30)
      Contact( #IO.HomeLimit )
      Move(in := 0, out1 => #IO."Step")
   END_RUNG
   // the same network as SCL:
   #IO.ParkedTimeoutFault := #ParkedTimer.Q OR (#IO.ParkedTimeoutFault AND NOT #IO.FaultReset);
   #ParkedTimer(IN := #IO."Step" = 30, PT := #ParkedTimeoutMS);   // TON
   IF (#IO."Step" = 30) AND #IO.HomeLimit THEN #IO."Step" := 0; END_IF;
END_REGION

REGION Network 10: Jog Pre-Start Warning
   RUNG wire#powerrail
      Contact( #IO.JogExtendCmd )
      wire#w1
      { S7_Templates := "SrcType := Int" } EQ_Contact(in1 := #IO."Step", in2 := 0)
      { S7_Templates := "SrcType := Int" } EQ_Contact(in1 := #IO.Mode, in2 := 2)
      Coil( #IO.JogPreStartSounder )
   END_RUNG
   RUNG wire#powerrail
      Contact( #IO.JogRetractCmd )
   END_RUNG wire#w1
   RUNG wire#powerrail
      Contact( #IO.JogExtendCmd )
      wire#w2
      { S7_Templates := "SrcType := Int" } EQ_Contact(in1 := #IO."Step", in2 := 0)
      { S7_Templates := "SrcType := Int" } EQ_Contact(in1 := #IO.Mode, in2 := 2)
      { S7_Templates := "time_type := Time" } #JogPreStartTimer.TON(pt := #JogWarningTimeMS, et =>)
   END_RUNG
   RUNG wire#powerrail
      Contact( #IO.JogRetractCmd )
   END_RUNG wire#w2
   // the same network as SCL:
   #IO.JogPreStartSounder := (#IO.JogExtendCmd OR #IO.JogRetractCmd) AND (#IO."Step" = 0) AND (#IO.Mode = 2);
   #JogPreStartTimer(IN := (#IO.JogExtendCmd OR #IO.JogRetractCmd) AND (#IO."Step" = 0) AND (#IO.Mode = 2),   // TON
                     PT := #JogWarningTimeMS);
END_REGION

REGION Network 11: Extend And Retract Demand
   // PressureHold gates ExtendDemand so a confirmed jam holds the ram in place rather than continuing to push (a hold per C-123, not a fault - it clears and driving resumes the instant pressure has cleared). Jog demand only arms after JogPreStartTimer.Q so a jog button press always gets the same audible pre-start warning as an auto cycle, never an instant unwarned move.
   RUNG wire#powerrail
      { S7_Templates := "SrcType := Int" } EQ_Contact(in1 := #IO."Step", in2 := 10)
      I_Contact( #PressureHold )
      wire#w1
      Coil( #ExtendDemand )
   END_RUNG
   RUNG wire#powerrail
      { S7_Templates := "SrcType := Int" } EQ_Contact(in1 := #IO."Step", in2 := 0)
      { S7_Templates := "SrcType := Int" } EQ_Contact(in1 := #IO.Mode, in2 := 2)
      Contact( #IO.JogExtendCmd )
      Contact( #JogPreStartTimer.Q )
   END_RUNG wire#w1
   RUNG wire#powerrail
      { S7_Templates := "SrcType := Int" } EQ_Contact(in1 := #IO."Step", in2 := 30)
      wire#w2
      Coil( #RetractDemand )
   END_RUNG
   RUNG wire#powerrail
      { S7_Templates := "SrcType := Int" } EQ_Contact(in1 := #IO."Step", in2 := 0)
      { S7_Templates := "SrcType := Int" } EQ_Contact(in1 := #IO.Mode, in2 := 2)
      Contact( #IO.JogRetractCmd )
      Contact( #JogPreStartTimer.Q )
   END_RUNG wire#w2
   // the same network as SCL:
   #ExtendDemand := ((#IO."Step" = 10) AND NOT #PressureHold) OR ((#IO."Step" = 0) AND (#IO.Mode = 2) AND #IO.JogExtendCmd AND #JogPreStartTimer.Q);
   #RetractDemand := (#IO."Step" = 30) OR ((#IO."Step" = 0) AND (#IO.Mode = 2) AND #IO.JogRetractCmd AND #JogPreStartTimer.Q);
END_REGION

REGION Network 12: Pump Demand
   RUNG wire#powerrail
      Contact( #ExtendDemand )
      wire#w1
      Coil( #PumpDemand )
   END_RUNG
   RUNG wire#powerrail
      Contact( #RetractDemand )
   END_RUNG wire#w1
   RUNG wire#powerrail
      Contact( #PumpDemand )
      wire#w2
      Coil( #PumpEverDemanded )
   END_RUNG
   RUNG wire#powerrail
      Contact( #PumpEverDemanded )
   END_RUNG wire#w2
   // the same network as SCL:
   #PumpDemand := #ExtendDemand OR #RetractDemand;
   #PumpEverDemanded := #PumpDemand OR #PumpEverDemanded;
END_REGION

REGION Network 13: Pump Run-On Timer And Output Commands
   // Off-delay built from TON+inversion, not TOF/TONR (C-406). PumpEverDemanded guards a cold-start gap: on power-up PumpDemand and the timer's Q are both initially false, which would read as 'run-on already elapsed' and skip straight to no-run. RunPowerPack stays on through the run-on tail even after demand drops, but the Extend/Retract solenoids are not - they only ever follow live demand, gated by PowerPackRunningFB so the ram can't be commanded before the pump has confirmed running.
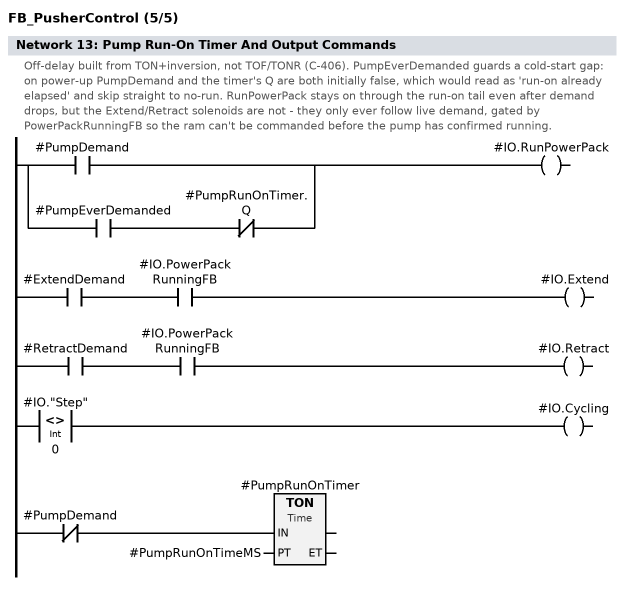
   RUNG wire#powerrail
      Contact( #PumpDemand )
      wire#w1
      Coil( #IO.RunPowerPack )
   END_RUNG
   RUNG wire#powerrail
      Contact( #PumpEverDemanded )
      I_Contact( #PumpRunOnTimer.Q )
   END_RUNG wire#w1
   RUNG wire#powerrail
      Contact( #ExtendDemand )
      Contact( #IO.PowerPackRunningFB )
      Coil( #IO.Extend )
   END_RUNG
   RUNG wire#powerrail
      Contact( #RetractDemand )
      Contact( #IO.PowerPackRunningFB )
      Coil( #IO.Retract )
   END_RUNG
   RUNG wire#powerrail
      { S7_Templates := "SrcType := Int" } NE_Contact(in1 := #IO."Step", in2 := 0)
      Coil( #IO.Cycling )
   END_RUNG
   RUNG wire#powerrail
      I_Contact( #PumpDemand )
      { S7_Templates := "time_type := Time" } #PumpRunOnTimer.TON(pt := #PumpRunOnTimeMS, et =>)
   END_RUNG
   // the same network as SCL:
   #IO.RunPowerPack := #PumpDemand OR (#PumpEverDemanded AND NOT #PumpRunOnTimer.Q);
   #IO.Extend := #ExtendDemand AND #IO.PowerPackRunningFB;
   #IO.Retract := #RetractDemand AND #IO.PowerPackRunningFB;
   #IO.Cycling := #IO."Step" <> 0;
   #PumpRunOnTimer(IN := NOT #PumpDemand, PT := #PumpRunOnTimeMS);   // TON
END_REGION
END_FUNCTION_BLOCK

FUNCTION "FC_Outputs" : Void   // FC2, LAD
TITLE = Output Map
{ S7_Optimized_Access := 'TRUE' }
VERSION : 0.1
// stored: AutoNumber true, IsIECCheckEnabled false, SetENOAutomatically false, UDAEnableTagReadback false
BEGIN

REGION Network 1: PLC1 Built-in DQ (CPU 1214C)
